C05480=1155.240,358.418,-80.283,-176.328,9.114,148.774
C05481=1155.245,358.171,-80.248,-176.331,9.110,148.773
C05482=1155.248,357.923,-80.214,-176.333,9.107,148.773
C05483=1155.252,357.676,-80.179,-176.336,9.102,148.773
C05484=1155.256,357.428,-80.144,-176.338,9.099,148.772
C05485=1155.261,357.181,-80.109,-176.341,9.095,148.772
C05486=1155.264,356.933,-80.075,-176.343,9.091,148.772
C05487=1155.268,356.685,-80.040,-176.345,9.087,148.771
C05488=1155.272,356.438,-80.005,-176.348,9.084,148.771
C05489=1155.276,356.190,-79.971,-176.350,9.080,148.771
C05490=1155.280,355.943,-79.937,-176.352,9.076,148.770
C05491=1155.284,355.695,-79.902,-176.355,9.072,148.770
C05492=1155.288,355.448,-79.868,-176.358,9.069,148.770
C05493=1155.292,355.200,-79.832,-176.360,9.065,148.770
C05494=1155.296,354.953,-79.798,-176.362,9.061,148.769
C05495=1155.299,354.705,-79.764,-176.365,9.057,148.769
C05496=1155.304,354.457,-79.729,-176.368,9.054,148.769
C05497=1155.308,354.210,-79.695,-176.370,9.049,148.768
C05498=1155.312,353.962,-79.660,-176.372,9.046,148.768
C05499=1155.316,353.715,-79.626,-176.375,9.042,148.768
C05500=1155.320,353.467,-79.592,-176.378,9.039,148.768
C05501=1155.324,353.220,-79.557,-176.380,9.034,148.767
C05502=1155.327,352.972,-79.523,-176.382,9.031,148.767
C05503=1155.332,352.724,-79.489,-176.385,9.027,148.767
C05504=1155.336,352.476,-79.454,-176.388,9.024,148.767
C05505=1155.340,352.229,-79.420,-176.390,9.019,148.766
C05506=1155.344,351.982,-79.385,-176.392,9.016,148.766
C05507=1155.348,351.734,-79.351,-176.395,9.012,148.766
C05508=1155.352,351.486,-79.317,-176.398,9.008,148.765
C05509=1155.355,351.239,-79.282,-176.400,9.004,148.765
C05510=1155.360,350.991,-79.248,-176.402,9.001,148.765
C05511=1155.364,350.744,-79.214,-176.405,8.997,148.764
C05512=1155.368,350.495,-79.180,-176.408,8.993,148.764
C05513=1155.372,350.248,-79.146,-176.410,8.989,148.764
C05514=1155.376,350.000,-79.111,-176.412,8.986,148.764
C05515=1155.380,349.753,-79.077,-176.415,8.982,148.763
C05516=1155.384,349.506,-79.043,-176.417,8.978,148.763
C05517=1155.388,349.257,-79.009,-176.420,8.974,148.763
C05518=1155.392,349.010,-78.976,-176.422,8.971,148.762
C05519=1155.396,348.763,-78.941,-176.425,8.967,148.762
C05520=1155.399,348.515,-78.907,-176.427,8.963,148.762
C05521=1155.404,348.267,-78.873,-176.430,8.960,148.762
C05522=1155.408,348.020,-78.839,-176.433,8.956,148.761
C05523=1155.411,347.772,-78.805,-176.435,8.952,148.761
C05524=1155.416,347.524,-78.771,-176.437,8.948,148.761
C05525=1155.420,347.277,-78.737,-176.440,8.945,148.761
C05526=1155.424,347.029,-78.703,-176.443,8.941,148.760
C05527=1155.428,346.781,-78.669,-176.445,8.938,148.760
C05528=1155.432,346.534,-78.635,-176.448,8.933,148.760
C05529=1155.436,346.286,-78.601,-176.450,8.930,148.759
C05530=1155.440,346.038,-78.567,-176.453,8.926,148.759
C05531=1155.444,345.791,-78.534,-176.455,8.922,148.759
C05532=1155.449,345.543,-78.500,-176.457,8.919,148.759
C05533=1155.452,345.295,-78.466,-176.460,8.915,148.759
C05534=1155.456,345.048,-78.432,-176.462,8.912,148.758
C05535=1155.461,344.800,-78.398,-176.465,8.907,148.758
C05536=1155.465,344.553,-78.364,-176.467,8.904,148.758
C05537=1155.468,344.304,-78.331,-176.470,8.900,148.757
C05538=1155.472,344.057,-78.297,-176.472,8.897,148.757
C05539=1155.477,343.809,-78.263,-176.475,8.893,148.757
C05540=1155.481,343.561,-78.230,-176.478,8.889,148.757
C05541=1155.484,343.314,-78.196,-176.480,8.886,148.757
C05542=1155.488,343.066,-78.162,-176.483,8.882,148.756
C05543=1155.493,342.818,-78.128,-176.485,8.879,148.756
C05544=1155.497,342.571,-78.095,-176.488,8.874,148.756
C05545=1155.501,342.323,-78.062,-176.490,8.871,148.755
C05546=1155.504,342.075,-78.027,-176.492,8.868,148.755
C05547=1155.509,341.827,-77.994,-176.495,8.864,148.755
C05548=1155.513,341.579,-77.961,-176.497,8.860,148.755
C05549=1155.517,341.332,-77.927,-176.500,8.856,148.755
C05550=1155.521,341.085,-77.894,-176.503,8.853,148.754
C05551=1155.526,340.837,-77.860,-176.505,8.850,148.754
C05552=1155.529,340.589,-77.826,-176.508,8.846,148.754
C05553=1155.533,340.341,-77.793,-176.510,8.842,148.754
C05554=1155.537,340.094,-77.760,-176.513,8.838,148.753
C05555=1155.542,339.814,-77.722,-176.516,8.834,148.753
C05556=1155.546,339.533,-77.684,-176.518,8.830,148.753
C05557=1155.551,339.254,-77.646,-176.521,8.826,148.752
C05558=1155.556,338.974,-77.609,-176.524,8.822,148.752
C05559=1155.560,338.727,-77.576,-176.527,8.818,148.752
C05560=1155.564,338.478,-77.541,-176.529,8.815,148.752
C05561=1155.568,338.230,-77.508,-176.532,8.811,148.752
C05562=1155.572,337.983,-77.474,-176.534,8.808,148.751
C05563=1155.576,337.735,-77.441,-176.536,8.804,148.751
C05564=1155.580,337.487,-77.408,-176.539,8.800,148.751
C05565=1155.584,337.240,-77.375,-176.542,8.797,148.751
C05566=1155.588,336.992,-77.342,-176.544,8.793,148.750
C05567=1155.593,336.744,-77.309,-176.547,8.790,148.750
C05568=1155.597,336.497,-77.275,-176.549,8.786,148.750
C05569=1155.600,336.248,-77.242,-176.552,8.782,148.750
C05570=1155.604,336.000,-77.209,-176.554,8.779,148.750
C05571=1155.608,335.753,-77.176,-176.557,8.776,148.749
C05572=1155.612,335.505,-77.143,-176.559,8.772,148.749
C05573=1155.616,335.258,-77.110,-176.562,8.768,148.749
C05574=1155.620,335.010,-77.077,-176.565,8.764,148.749
C05575=1155.624,334.762,-77.044,-176.567,8.761,148.749
C05576=1155.629,334.514,-77.010,-176.569,8.758,148.748
C05577=1155.633,334.267,-76.977,-176.572,8.753,148.748
C05578=1155.637,334.019,-76.944,-176.575,8.750,148.748
C05579=1155.641,333.771,-76.911,-176.577,8.747,148.748
C05580=1155.645,333.523,-76.879,-176.580,8.743,148.747
C05581=1155.649,333.275,-76.846,-176.582,8.740,148.747
C05582=1155.653,333.028,-76.813,-176.584,8.736,148.747
C05583=1155.657,332.780,-76.780,-176.587,8.732,148.747
C05584=1155.661,332.532,-76.747,-176.590,8.729,148.747
C05585=1155.665,332.284,-76.713,-176.592,8.726,148.746
C05586=1155.670,332.036,-76.681,-176.595,8.722,148.746
C05587=1155.673,331.789,-76.648,-176.597,8.718,148.746
C05588=1155.677,331.541,-76.615,-176.599,8.715,148.746
C05589=1155.681,331.293,-76.582,-176.603,8.711,148.746
C05590=1155.686,331.045,-76.550,-176.605,8.708,148.745
C05591=1155.690,330.797,-76.516,-176.608,8.704,148.745
C05592=1155.693,330.550,-76.484,-176.610,8.701,148.745
C05593=1155.698,330.301,-76.451,-176.613,8.697,148.745
C05594=1155.702,330.054,-76.418,-176.615,8.693,148.745
C05595=1155.706,329.806,-76.385,-176.618,8.690,148.744
C05596=1155.710,329.558,-76.353,-176.620,8.687,148.744
C05597=1155.714,329.310,-76.320,-176.622,8.683,148.744
C05598=1155.719,329.063,-76.287,-176.625,8.679,148.744
C05599=1155.723,328.815,-76.255,-176.628,8.676,148.744
C05600=1155.727,328.567,-76.222,-176.630,8.673,148.743
C05601=1155.731,328.319,-76.190,-176.633,8.669,148.743
C05602=1155.735,328.071,-76.157,-176.636,8.666,148.743
C05603=1155.739,327.824,-76.124,-176.638,8.662,148.743
C05604=1155.743,327.576,-76.092,-176.641,8.658,148.743
C05605=1155.747,327.328,-76.059,-176.643,8.655,148.743
C05606=1155.751,327.080,-76.027,-176.645,8.652,148.742
C05607=1155.756,326.833,-75.994,-176.648,8.648,148.742
C05608=1155.760,326.584,-75.962,-176.651,8.644,148.742
C05609=1155.763,326.337,-75.929,-176.653,8.641,148.742
C05610=1155.768,326.089,-75.897,-176.656,8.637,148.742
C05611=1155.772,325.841,-75.865,-176.658,8.634,148.741
C05612=1155.776,325.593,-75.832,-176.661,8.631,148.741
C05613=1155.780,325.344,-75.799,-176.663,8.627,148.741
C05614=1155.784,325.098,-75.767,-176.666,8.623,148.741
C05615=1155.789,324.849,-75.734,-176.668,8.620,148.741
C05616=1155.792,324.601,-75.703,-176.671,8.617,148.740
C05617=1155.796,324.354,-75.669,-176.674,8.613,148.740
C05618=1155.800,324.106,-75.638,-176.676,8.610,148.740
C05619=1155.805,323.857,-75.605,-176.679,8.606,148.740
C05620=1155.809,323.611,-75.573,-176.681,8.602,148.740
C05621=1155.813,323.362,-75.541,-176.684,8.599,148.740
C05622=1155.817,323.114,-75.509,-176.686,8.596,148.739
C05623=1155.821,322.866,-75.476,-176.689,8.593,148.739
C05624=1155.825,322.618,-75.444,-176.692,8.589,148.739
C05625=1155.830,322.371,-75.412,-176.694,8.585,148.739
C05626=1155.833,322.123,-75.380,-176.696,8.582,148.739
C05627=1155.838,321.874,-75.347,-176.699,8.578,148.739
C05628=1155.841,321.627,-75.315,-176.702,8.575,148.739
C05629=1155.846,321.380,-75.283,-176.704,8.572,148.738
C05630=1155.850,321.131,-75.251,-176.707,8.568,148.738
C05631=1155.854,320.883,-75.219,-176.710,8.564,148.738
C05632=1155.858,320.635,-75.187,-176.712,8.561,148.738
C05633=1155.862,320.388,-75.155,-176.715,8.558,148.738
C05634=1155.866,320.140,-75.123,-176.717,8.555,148.738
C05635=1155.870,319.892,-75.090,-176.720,8.551,148.737
C05636=1155.874,319.644,-75.058,-176.722,8.548,148.737
C05637=1155.879,319.396,-75.026,-176.725,8.545,148.737
C05638=1155.883,319.148,-74.994,-176.727,8.541,148.737
C05639=1155.886,318.900,-74.962,-176.730,8.537,148.737
C05640=1155.891,318.652,-74.930,-176.732,8.534,148.737
C05641=1155.895,318.404,-74.899,-176.735,8.531,148.736
C05642=1155.899,318.156,-74.867,-176.738,8.527,148.736
C05643=1155.903,317.908,-74.834,-176.740,8.524,148.736
C05644=1155.908,317.661,-74.803,-176.743,8.520,148.736
C05645=1155.911,317.413,-74.771,-176.745,8.517,148.736
C05646=1155.915,317.164,-74.739,-176.748,8.513,148.736
C05647=1155.920,316.917,-74.707,-176.751,8.510,148.736
C05648=1155.924,316.669,-74.675,-176.753,8.507,148.735
C05649=1155.927,316.421,-74.643,-176.756,8.504,148.735
C05650=1155.932,316.173,-74.613,-176.759,8.500,148.735
C05651=1155.937,315.924,-74.580,-176.761,8.496,148.735
C05652=1155.941,315.677,-74.549,-176.763,8.493,148.735
C05653=1155.945,315.429,-74.517,-176.766,8.490,148.735
C05654=1155.948,315.181,-74.485,-176.768,8.487,148.735
C05655=1155.953,314.933,-74.453,-176.771,8.483,148.734
C05656=1155.957,314.685,-74.422,-176.773,8.479,148.734
C05657=1155.961,314.437,-74.390,-176.776,8.476,148.734
C05658=1155.965,314.189,-74.358,-176.778,8.473,148.734
C05659=1155.970,313.912,-74.323,-176.781,8.469,148.734
C05660=1155.975,313.635,-74.288,-176.785,8.465,148.734
C05661=1155.979,313.357,-74.253,-176.788,8.461,148.734
C05662=1155.984,313.079,-74.217,-176.790,8.458,148.733
C05663=1155.988,312.832,-74.186,-176.793,8.454,148.733
C05664=1155.992,312.584,-74.153,-176.796,8.451,148.733
C05665=1155.997,312.336,-74.122,-176.798,8.448,148.733
C05666=1156.001,312.088,-74.091,-176.801,8.445,148.733
C05667=1156.005,311.840,-74.059,-176.803,8.441,148.733
C05668=1156.009,311.592,-74.028,-176.806,8.437,148.733
C05669=1156.013,311.344,-73.996,-176.809,8.434,148.733
C05670=1156.017,311.096,-73.965,-176.811,8.431,148.732
C05671=1156.022,310.848,-73.934,-176.813,8.428,148.732
C05672=1156.025,310.600,-73.902,-176.816,8.425,148.732
C05673=1156.030,310.352,-73.871,-176.819,8.421,148.732
C05674=1156.034,310.104,-73.839,-176.821,8.417,148.732
C05675=1156.038,309.856,-73.808,-176.824,8.414,148.732
C05676=1156.042,309.608,-73.777,-176.826,8.411,148.732
C05677=1156.047,309.360,-73.745,-176.829,8.408,148.732
C05678=1156.051,309.112,-73.714,-176.832,8.404,148.731
C05679=1156.056,308.864,-73.683,-176.834,8.401,148.731
C05680=1156.059,308.616,-73.651,-176.837,8.398,148.731
C05681=1156.064,308.368,-73.620,-176.839,8.395,148.731
C05682=1156.067,308.120,-73.590,-176.842,8.391,148.731
C05683=1156.071,307.872,-73.558,-176.845,8.388,148.731
C05684=1156.075,307.624,-73.527,-176.847,8.384,148.731
C05685=1156.080,307.376,-73.496,-176.850,8.381,148.731
C05686=1156.084,307.128,-73.464,-176.852,8.378,148.731
C05687=1156.088,306.880,-73.434,-176.855,8.375,148.730
C05688=1156.092,306.632,-73.402,-176.858,8.371,148.730
C05689=1156.097,306.384,-73.371,-176.860,8.368,148.730
C05690=1156.101,306.136,-73.340,-176.863,8.365,148.730
C05691=1156.105,305.888,-73.308,-176.865,8.361,148.730
C05692=1156.110,305.640,-73.278,-176.868,8.358,148.730
C05693=1156.114,305.391,-73.247,-176.871,8.354,148.730
C05694=1156.118,305.144,-73.215,-176.873,8.351,148.730
C05695=1156.122,304.896,-73.185,-176.876,8.348,148.730
C05696=1156.126,304.647,-73.154,-176.878,8.345,148.729
C05697=1156.130,304.400,-73.123,-176.881,8.342,148.729
C05698=1156.134,304.151,-73.092,-176.883,8.339,148.729
C05699=1156.139,303.904,-73.060,-176.886,8.335,148.729
C05700=1156.143,303.656,-73.030,-176.889,8.332,148.729
C05701=1156.147,303.407,-72.999,-176.891,8.328,148.729
C05702=1156.151,303.159,-72.968,-176.894,8.325,148.729
C05703=1156.156,302.911,-72.938,-176.896,8.322,148.729
C05704=1156.160,302.663,-72.906,-176.899,8.319,148.729
C05705=1156.164,302.415,-72.875,-176.902,8.315,148.729
C05706=1156.168,302.168,-72.845,-176.904,8.312,148.728
C05707=1156.172,301.919,-72.814,-176.907,8.309,148.728
C05708=1156.177,301.671,-72.783,-176.909,8.306,148.728
C05709=1156.181,301.423,-72.752,-176.912,8.303,148.728
C05710=1156.185,301.175,-72.722,-176.915,8.299,148.728
C05711=1156.189,300.927,-72.691,-176.917,8.296,148.728
C05712=1156.194,300.679,-72.660,-176.920,8.292,148.728
C05713=1156.197,300.430,-72.630,-176.923,8.289,148.728
C05714=1156.202,300.183,-72.599,-176.925,8.286,148.728
C05715=1156.206,299.935,-72.568,-176.928,8.283,148.728
C05716=1156.210,299.687,-72.538,-176.930,8.280,148.728
C05717=1156.214,299.438,-72.507,-176.933,8.277,148.728
C05718=1156.219,299.190,-72.476,-176.935,8.274,148.727
C05719=1156.223,298.943,-72.446,-176.939,8.270,148.727
C05720=1156.227,298.695,-72.415,-176.941,8.266,148.727
C05721=1156.232,298.445,-72.385,-176.944,8.263,148.727
C05722=1156.236,298.198,-72.354,-176.946,8.260,148.727
C05723=1156.240,297.950,-72.324,-176.949,8.257,148.727
C05724=1156.245,297.702,-72.293,-176.951,8.254,148.727
C05725=1156.248,297.453,-72.262,-176.954,8.251,148.727
C05726=1156.253,297.206,-72.232,-176.957,8.247,148.727
C05727=1156.257,296.957,-72.202,-176.960,8.244,148.727
C05728=1156.261,296.709,-72.171,-176.962,8.241,148.727
C05729=1156.265,296.461,-72.141,-176.965,8.238,148.727
C05730=1156.269,296.213,-72.110,-176.967,8.234,148.727
C05731=1156.273,295.965,-72.080,-176.970,8.232,148.727
C05732=1156.278,295.717,-72.050,-176.972,8.228,148.726
C05733=1156.283,295.469,-72.019,-176.975,8.225,148.726
C05734=1156.286,295.220,-71.989,-176.978,8.222,148.726
C05735=1156.291,294.972,-71.959,-176.980,8.218,148.726
C05736=1156.295,294.724,-71.928,-176.983,8.215,148.726
C05737=1156.299,294.477,-71.898,-176.986,8.212,148.726
C05738=1156.304,294.228,-71.868,-176.988,8.209,148.726
C05739=1156.307,293.980,-71.838,-176.991,8.206,148.726
C05740=1156.311,293.732,-71.807,-176.993,8.203,148.726
C05741=1156.316,293.483,-71.777,-176.996,8.200,148.726
C05742=1156.320,293.235,-71.747,-176.998,8.197,148.726
C05743=1156.324,292.988,-71.716,-177.002,8.193,148.726
C05744=1156.329,292.739,-71.686,-177.004,8.190,148.726
C05745=1156.333,292.492,-71.656,-177.007,8.187,148.726
C05746=1156.337,292.243,-71.626,-177.009,8.183,148.726
C05747=1156.341,291.995,-71.596,-177.012,8.180,148.726
C05748=1156.345,291.746,-71.566,-177.014,8.177,148.725
C05749=1156.350,291.498,-71.535,-177.017,8.174,148.725
C05750=1156.354,291.250,-71.506,-177.020,8.171,148.725
C05751=1156.358,291.003,-71.476,-177.022,8.168,148.725
C05752=1156.363,290.754,-71.446,-177.025,8.165,148.725
C05753=1156.367,290.506,-71.416,-177.028,8.161,148.725
C05754=1156.371,290.258,-71.386,-177.030,8.158,148.725
C05755=1156.375,290.009,-71.355,-177.033,8.155,148.725
C05756=1156.379,289.761,-71.326,-177.036,8.152,148.725
C05757=1156.383,289.513,-71.296,-177.038,8.149,148.725
C05758=1156.388,289.265,-71.265,-177.041,8.146,148.725
C05759=1156.392,289.017,-71.236,-177.043,8.142,148.725
C05760=1156.396,288.769,-71.206,-177.046,8.139,148.725
C05761=1156.400,288.521,-71.176,-177.048,8.136,148.725
C05762=1156.405,288.272,-71.146,-177.051,8.133,148.725
C05763=1156.410,287.997,-71.113,-177.055,8.129,148.725
C05764=1156.415,287.722,-71.080,-177.057,8.126,148.725
C05765=1156.419,287.447,-71.047,-177.060,8.122,148.725
C05766=1156.424,287.172,-71.014,-177.063,8.119,148.725
C05767=1156.428,286.924,-70.984,-177.066,8.117,148.725
C05768=1156.432,286.676,-70.955,-177.068,8.113,148.725
C05769=1156.437,286.428,-70.925,-177.071,8.109,148.725
C05770=1156.441,286.179,-70.895,-177.074,8.107,148.725
C05771=1156.446,285.931,-70.866,-177.076,8.103,148.724
C05772=1156.450,285.683,-70.836,-177.079,8.100,148.724
C05773=1156.454,285.435,-70.806,-177.082,8.097,148.725
C05774=1156.458,285.187,-70.777,-177.084,8.094,148.724
C05775=1156.462,284.938,-70.747,-177.087,8.091,148.724
C05776=1156.467,284.690,-70.717,-177.090,8.088,148.724
C05777=1156.471,284.442,-70.688,-177.092,8.085,148.724
C05778=1156.475,284.193,-70.658,-177.095,8.082,148.724
C05779=1156.479,283.946,-70.628,-177.098,8.079,148.724
C05780=1156.483,283.697,-70.599,-177.100,8.076,148.724
C05781=1156.488,283.449,-70.569,-177.103,8.073,148.724
C05782=1156.492,283.201,-70.540,-177.105,8.070,148.724
C05783=1156.496,282.953,-70.510,-177.108,8.067,148.724
C05784=1156.500,282.704,-70.481,-177.111,8.064,148.724
C05785=1156.505,282.456,-70.451,-177.113,8.061,148.724
C05786=1156.509,282.207,-70.421,-177.116,8.057,148.724
C05787=1156.513,281.959,-70.392,-177.118,8.054,148.724
C05788=1156.518,281.712,-70.363,-177.122,8.051,148.724
C05789=1156.522,281.463,-70.333,-177.124,8.048,148.724
C05790=1156.527,281.215,-70.304,-177.127,8.044,148.724
C05791=1156.531,280.967,-70.275,-177.130,8.041,148.724
C05792=1156.535,280.718,-70.246,-177.132,8.038,148.724
C05793=1156.539,280.470,-70.216,-177.135,8.036,148.724
C05794=1156.544,280.221,-70.187,-177.137,8.032,148.724
C05795=1156.548,279.973,-70.157,-177.140,8.029,148.724
C05796=1156.553,279.726,-70.128,-177.143,8.026,148.724
C05797=1156.557,279.477,-70.099,-177.145,8.023,148.724
C05798=1156.561,279.229,-70.069,-177.148,8.020,148.724
C05799=1156.565,278.981,-70.040,-177.151,8.017,148.724
C05800=1156.569,278.732,-70.012,-177.154,8.014,148.724
C05801=1156.573,278.484,-69.982,-177.156,8.011,148.724
C05802=1156.578,278.236,-69.953,-177.159,8.008,148.724
C05803=1156.582,277.988,-69.924,-177.161,8.005,148.724
C05804=1156.586,277.739,-69.895,-177.164,8.002,148.724
C05805=1156.591,277.491,-69.866,-177.166,7.999,148.724
C05806=1156.595,277.243,-69.836,-177.169,7.996,148.724
C05807=1156.599,276.994,-69.807,-177.172,7.993,148.724
C05808=1156.604,276.746,-69.778,-177.175,7.990,148.724
C05809=1156.608,276.498,-69.749,-177.177,7.987,148.724
C05810=1156.612,276.250,-69.720,-177.180,7.984,148.724
C05811=1156.616,276.001,-69.691,-177.183,7.981,148.724
C05812=1156.620,275.753,-69.662,-177.185,7.978,148.724
C05813=1156.625,275.505,-69.633,-177.188,7.975,148.724
C05814=1156.629,275.257,-69.605,-177.190,7.972,148.724
C05815=1156.633,275.008,-69.575,-177.193,7.969,148.724
C05816=1156.638,274.759,-69.546,-177.196,7.966,148.724
C05817=1156.642,274.512,-69.517,-177.199,7.963,148.724
C05818=1156.647,274.264,-69.488,-177.201,7.960,148.724
C05819=1156.650,274.015,-69.460,-177.204,7.957,148.724
C05820=1156.654,273.767,-69.430,-177.207,7.954,148.724
C05821=1156.660,273.519,-69.402,-177.209,7.951,148.724
C05822=1156.664,273.270,-69.372,-177.212,7.948,148.724
C05823=1156.668,273.022,-69.344,-177.215,7.945,148.724
C05824=1156.672,272.774,-69.315,-177.218,7.942,148.724
C05825=1156.677,272.525,-69.287,-177.220,7.939,148.724
C05826=1156.680,272.277,-69.258,-177.223,7.936,148.724
C05827=1156.685,272.029,-69.229,-177.225,7.933,148.724
C05828=1156.690,271.780,-69.201,-177.228,7.930,148.724
C05829=1156.694,271.532,-69.171,-177.231,7.927,148.724
C05830=1156.698,271.283,-69.143,-177.234,7.924,148.724
C05831=1156.703,271.036,-69.114,-177.236,7.921,148.724
C05832=1156.706,270.787,-69.086,-177.239,7.918,148.724
C05833=1156.711,270.538,-69.057,-177.242,7.915,148.724
C05834=1156.716,270.291,-69.028,-177.244,7.912,148.724
C05835=1156.719,270.042,-69.000,-177.247,7.909,148.724
C05836=1156.724,269.794,-68.971,-177.250,7.906,148.724
C05837=1156.729,269.546,-68.942,-177.252,7.902,148.724
C05838=1156.732,269.297,-68.914,-177.255,7.900,148.724
C05839=1156.737,269.049,-68.885,-177.258,7.897,148.724
C05840=1156.741,268.800,-68.857,-177.260,7.894,148.724
C05841=1156.745,268.552,-68.828,-177.263,7.891,148.724
C05842=1156.750,268.304,-68.799,-177.265,7.889,148.724
C05843=1156.754,268.055,-68.771,-177.268,7.886,148.724
C05844=1156.759,267.807,-68.743,-177.271,7.883,148.725
C05845=1156.763,267.559,-68.714,-177.273,7.879,148.724
C05846=1156.767,267.310,-68.685,-177.276,7.876,148.724
C05847=1156.772,267.063,-68.658,-177.279,7.874,148.724
C05848=1156.776,266.814,-68.629,-177.282,7.871,148.725
C05849=1156.780,266.566,-68.601,-177.284,7.868,148.725
C05850=1156.785,266.317,-68.572,-177.287,7.865,148.725
C05851=1156.789,266.070,-68.544,-177.290,7.862,148.725
C05852=1156.793,265.821,-68.515,-177.293,7.859,148.725
C05853=1156.797,265.572,-68.487,-177.295,7.856,148.725
C05854=1156.802,265.324,-68.459,-177.298,7.853,148.725
C05855=1156.806,265.075,-68.430,-177.301,7.850,148.725
C05856=1156.811,264.827,-68.402,-177.303,7.847,148.725
C05857=1156.815,264.579,-68.374,-177.306,7.844,148.725
C05858=1156.820,264.330,-68.346,-177.309,7.841,148.725
C05859=1156.824,264.082,-68.317,-177.312,7.838,148.725
C05860=1156.828,263.834,-68.290,-177.314,7.835,148.725
C05861=1156.832,263.585,-68.261,-177.317,7.833,148.725
C05862=1156.837,263.337,-68.233,-177.319,7.830,148.725
C05863=1156.841,263.088,-68.204,-177.322,7.827,148.725
C05864=1156.846,262.840,-68.177,-177.325,7.824,148.725
C05865=1156.849,262.592,-68.148,-177.328,7.821,148.725
C05866=1156.855,262.344,-68.120,-177.330,7.818,148.725
C05867=1156.859,262.070,-68.089,-177.333,7.815,148.725
C05868=1156.864,261.797,-68.059,-177.337,7.811,148.725
C05869=1156.869,261.524,-68.028,-177.339,7.808,148.725
C05870=1156.873,261.250,-67.997,-177.342,7.805,148.726
C05871=1156.878,261.002,-67.969,-177.345,7.802,148.726
C05872=1156.882,260.754,-67.941,-177.348,7.800,148.726
C05873=1156.886,260.506,-67.913,-177.350,7.797,148.726
C05874=1156.891,260.257,-67.884,-177.353,7.794,148.726
C05875=1156.896,260.008,-67.857,-177.356,7.791,148.726
C05876=1156.899,259.760,-67.829,-177.359,7.788,148.726
C05877=1156.904,259.512,-67.801,-177.361,7.785,148.726
C05878=1156.908,259.263,-67.773,-177.364,7.782,148.726
C05879=1156.913,259.015,-67.746,-177.366,7.779,148.726
C05880=1156.917,258.767,-67.718,-177.369,7.776,148.726
C05881=1156.921,258.518,-67.690,-177.371,7.774,148.726
C05882=1156.926,258.269,-67.662,-177.374,7.771,148.726
C05883=1156.930,258.021,-67.634,-177.377,7.768,148.726
C05884=1156.934,257.773,-67.606,-177.380,7.765,148.726
C05885=1156.939,257.524,-67.579,-177.383,7.762,148.726
C05886=1156.943,257.276,-67.551,-177.385,7.759,148.726
C05887=1156.948,257.028,-67.522,-177.388,7.756,148.726
C05888=1156.952,256.778,-67.495,-177.391,7.753,148.726
C05889=1156.956,256.530,-67.467,-177.393,7.751,148.727
C05890=1156.961,256.283,-67.439,-177.396,7.748,148.727
C05891=1156.965,256.033,-67.412,-177.399,7.745,148.727
C05892=1156.969,255.786,-67.384,-177.401,7.742,148.727
C05893=1156.974,255.537,-67.357,-177.404,7.739,148.727
C05894=1156.978,255.288,-67.328,-177.407,7.736,148.727
C05895=1156.983,255.040,-67.301,-177.410,7.733,148.727
C05896=1156.987,254.792,-67.274,-177.412,7.730,148.727
C05897=1156.991,254.543,-67.246,-177.415,7.728,148.727
C05898=1156.996,254.295,-67.218,-177.418,7.725,148.727
C05899=1157.000,254.046,-67.191,-177.421,7.722,148.727
C05900=1157.005,253.798,-67.164,-177.423,7.720,148.728
C05901=1157.009,253.549,-67.136,-177.426,7.717,148.728
C05902=1157.013,253.301,-67.108,-177.429,7.714,148.728
C05903=1157.018,253.053,-67.081,-177.432,7.711,148.728
C05904=1157.022,252.804,-67.054,-177.434,7.708,148.728
C05905=1157.026,252.556,-67.026,-177.437,7.706,148.728
C05906=1157.031,252.307,-66.999,-177.439,7.703,148.728
C05907=1157.035,252.059,-66.971,-177.442,7.700,148.728
C05908=1157.039,251.810,-66.944,-177.445,7.697,148.728
C05909=1157.044,251.562,-66.917,-177.448,7.694,148.728
C05910=1157.048,251.314,-66.889,-177.451,7.691,148.728
C05911=1157.053,251.065,-66.862,-177.453,7.688,148.728
C05912=1157.057,250.816,-66.835,-177.456,7.686,148.728
C05913=1157.061,250.568,-66.807,-177.458,7.683,148.728
C05914=1157.066,250.320,-66.780,-177.461,7.680,148.728
C05915=1157.070,250.071,-66.753,-177.464,7.677,148.729
C05916=1157.075,249.822,-66.725,-177.467,7.674,148.729
C05917=1157.079,249.574,-66.697,-177.470,7.672,148.729
C05918=1157.084,249.326,-66.670,-177.472,7.669,148.729
C05919=1157.088,249.077,-66.643,-177.475,7.666,148.729
C05920=1157.092,248.829,-66.617,-177.478,7.664,148.729
C05921=1157.096,248.580,-66.589,-177.480,7.661,148.729
C05922=1157.101,248.332,-66.562,-177.483,7.658,148.729
C05923=1157.105,248.083,-66.535,-177.486,7.655,148.729
C05924=1157.110,247.835,-66.508,-177.488,7.653,148.729
C05925=1157.115,247.586,-66.480,-177.491,7.650,148.730
C05926=1157.119,247.338,-66.453,-177.494,7.647,148.730
C05927=1157.122,247.089,-66.427,-177.497,7.644,148.730
C05928=1157.127,246.841,-66.399,-177.500,7.641,148.730
C05929=1157.132,246.592,-66.372,-177.502,7.638,148.730
C05930=1157.136,246.344,-66.345,-177.505,7.636,148.730
C05931=1157.141,246.095,-66.318,-177.507,7.633,148.730
C05932=1157.145,245.847,-66.291,-177.510,7.630,148.730
C05933=1157.149,245.599,-66.264,-177.513,7.627,148.730
C05934=1157.153,245.350,-66.237,-177.516,7.624,148.730
C05935=1157.158,245.101,-66.210,-177.518,7.623,148.731
C05936=1157.162,244.853,-66.183,-177.521,7.620,148.731
C05937=1157.167,244.605,-66.156,-177.524,7.617,148.731
C05938=1157.172,244.355,-66.130,-177.527,7.614,148.731
C05939=1157.176,244.107,-66.103,-177.529,7.611,148.731
C05940=1157.180,243.859,-66.076,-177.532,7.609,148.731
C05941=1157.185,243.610,-66.049,-177.534,7.606,148.731
C05942=1157.190,243.362,-66.022,-177.538,7.603,148.731
C05943=1157.193,243.113,-65.995,-177.540,7.600,148.732
C05944=1157.197,242.864,-65.968,-177.543,7.597,148.732
C05945=1157.202,242.616,-65.941,-177.545,7.595,148.732
C05946=1157.207,242.367,-65.914,-177.548,7.592,148.732
C05947=1157.211,242.119,-65.888,-177.551,7.589,148.732
C05948=1157.216,241.870,-65.861,-177.554,7.586,148.732
C05949=1157.220,241.622,-65.835,-177.557,7.584,148.732
C05950=1157.224,241.373,-65.808,-177.559,7.582,148.732
C05951=1157.229,241.125,-65.781,-177.562,7.579,148.732
C05952=1157.233,240.877,-65.754,-177.565,7.576,148.732
C05953=1157.238,240.628,-65.728,-177.567,7.573,148.733
C05954=1157.242,240.379,-65.701,-177.570,7.570,148.733
C05955=1157.246,240.131,-65.674,-177.573,7.568,148.733
C05956=1157.251,239.883,-65.647,-177.576,7.565,148.733
C05957=1157.255,239.634,-65.621,-177.578,7.562,148.733
C05958=1157.260,239.385,-65.594,-177.581,7.559,148.733
C05959=1157.264,239.137,-65.568,-177.583,7.557,148.733
C05960=1157.269,238.888,-65.542,-177.587,7.554,148.734
C05961=1157.273,238.639,-65.515,-177.589,7.552,148.734
C05962=1157.277,238.391,-65.488,-177.592,7.549,148.734
C05963=1157.282,238.142,-65.462,-177.594,7.546,148.734
C05964=1157.286,237.894,-65.435,-177.597,7.544,148.734
C05965=1157.291,237.645,-65.409,-177.600,7.541,148.734
C05966=1157.295,237.397,-65.382,-177.603,7.538,148.734
C05967=1157.300,237.148,-65.355,-177.605,7.536,148.734
C05968=1157.304,236.899,-65.330,-177.608,7.533,148.734
C05969=1157.309,236.651,-65.303,-177.611,7.530,148.735
C05970=1157.313,236.402,-65.277,-177.614,7.527,148.735
C05971=1157.318,236.130,-65.247,-177.617,7.524,148.735
C05972=1157.322,235.859,-65.219,-177.620,7.522,148.735
C05973=1157.328,235.587,-65.190,-177.623,7.519,148.735
C05974=1157.332,235.316,-65.161,-177.626,7.516,148.735
C05975=1157.336,235.067,-65.136,-177.629,7.513,148.735
C05976=1157.341,234.818,-65.109,-177.631,7.510,148.736
C05977=1157.346,234.570,-65.083,-177.634,7.508,148.736
C05978=1157.351,234.322,-65.056,-177.637,7.505,148.736
C05979=1157.355,234.073,-65.030,-177.640,7.502,148.736
C05980=1157.359,233.824,-65.005,-177.642,7.500,148.736
C05981=1157.364,233.576,-64.978,-177.645,7.498,148.736
C05982=1157.368,233.327,-64.952,-177.648,7.495,148.737
C05983=1157.372,233.079,-64.925,-177.651,7.492,148.737
C05984=1157.377,232.830,-64.899,-177.653,7.490,148.737
C05985=1157.382,232.581,-64.874,-177.656,7.487,148.737
C05986=1157.386,232.333,-64.847,-177.659,7.484,148.737
C05987=1157.391,232.084,-64.821,-177.662,7.481,148.737
C05988=1157.395,231.835,-64.795,-177.664,7.479,148.737
C05989=1157.399,231.587,-64.769,-177.667,7.477,148.738
C05990=1157.404,231.338,-64.742,-177.670,7.474,148.738
C05991=1157.408,231.090,-64.717,-177.672,7.472,148.738
C05992=1157.413,230.841,-64.691,-177.675,7.469,148.738
C05993=1157.418,230.592,-64.665,-177.678,7.466,148.738
C05994=1157.422,230.344,-64.638,-177.681,7.463,148.738
C05995=1157.426,230.095,-64.612,-177.683,7.461,148.738
C05996=1157.431,229.847,-64.587,-177.686,7.458,148.739
C05997=1157.436,229.598,-64.561,-177.689,7.455,148.739
C05998=1157.439,229.350,-64.534,-177.691,7.453,148.739
C05999=1157.444,229.101,-64.509,-177.694,7.451,148.739
C06000=1157.448,228.852,-64.483,-177.697,7.448,148.739
C06001=1157.453,228.604,-64.457,-177.699,7.446,148.739
C06002=1157.458,228.355,-64.431,-177.702,7.443,148.739
C06003=1157.462,228.106,-64.405,-177.705,7.440,148.740
C06004=1157.466,227.857,-64.380,-177.708,7.438,148.740
C06005=1157.471,227.609,-64.354,-177.710,7.435,148.740
C06006=1157.475,227.360,-64.328,-177.714,7.432,148.740
C06007=1157.479,227.112,-64.302,-177.716,7.430,148.740
C06008=1157.483,226.863,-64.276,-177.719,7.427,148.740
C06009=1157.489,226.615,-64.250,-177.722,7.425,148.741
C06010=1157.493,226.366,-64.224,-177.725,7.422,148.741
C06011=1157.497,226.117,-64.199,-177.727,7.420,148.741
C06012=1157.502,225.868,-64.173,-177.730,7.417,148.741
C06013=1157.506,225.620,-64.148,-177.733,7.414,148.741
C06014=1157.511,225.372,-64.122,-177.735,7.412,148.741
C06015=1157.515,225.123,-64.096,-177.738,7.409,148.741
C06016=1157.520,224.875,-64.071,-177.741,7.407,148.742
C06017=1157.524,224.625,-64.046,-177.743,7.404,148.742
C06018=1157.528,224.376,-64.020,-177.746,7.402,148.742
C06019=1157.533,224.128,-63.995,-177.749,7.399,148.742
C06020=1157.538,223.879,-63.969,-177.752,7.397,148.742
C06021=1157.542,223.630,-63.942,-177.755,7.394,148.743
C06022=1157.547,223.382,-63.917,-177.758,7.391,148.743
C06023=1157.552,223.133,-63.891,-177.760,7.389,148.743
C06024=1157.556,222.885,-63.866,-177.763,7.387,148.743
C06025=1157.561,222.636,-63.841,-177.765,7.384,148.743
C06026=1157.565,222.387,-63.815,-177.768,7.382,148.743
C06027=1157.569,222.138,-63.789,-177.771,7.379,148.744
C06028=1157.574,221.890,-63.764,-177.773,7.377,148.744
C06029=1157.578,221.642,-63.739,-177.776,7.374,148.744
C06030=1157.583,221.393,-63.714,-177.779,7.371,148.744
C06031=1157.587,221.144,-63.688,-177.782,7.369,148.744
C06032=1157.591,220.895,-63.663,-177.784,7.366,148.744
C06033=1157.596,220.647,-63.637,-177.788,7.364,148.745
C06034=1157.601,220.398,-63.612,-177.790,7.362,148.745
C06035=1157.605,220.150,-63.587,-177.793,7.359,148.745
C06036=1157.610,219.901,-63.561,-177.795,7.357,148.745
C06037=1157.614,219.652,-63.536,-177.798,7.354,148.745
C06038=1157.619,219.403,-63.511,-177.801,7.351,148.746
C06039=1157.623,219.155,-63.485,-177.804,7.349,148.746
C06040=1157.628,218.906,-63.461,-177.806,7.346,148.746
C06041=1157.632,218.657,-63.435,-177.809,7.345,148.746
C06042=1157.637,218.409,-63.410,-177.812,7.342,148.746
C06043=1157.641,218.160,-63.385,-177.815,7.339,148.747
C06044=1157.645,217.911,-63.359,-177.817,7.337,148.747
C06045=1157.651,217.662,-63.334,-177.820,7.334,148.747
C06046=1157.654,217.414,-63.309,-177.823,7.331,148.747
C06047=1157.659,217.166,-63.284,-177.826,7.329,148.747
C06048=1157.663,216.916,-63.259,-177.829,7.327,148.748
C06049=1157.668,216.668,-63.233,-177.831,7.325,148.748
C06050=1157.673,216.419,-63.208,-177.834,7.322,148.748
C06051=1157.677,216.171,-63.183,-177.836,7.320,148.748
C06052=1157.681,215.922,-63.158,-177.839,7.317,148.748
C06053=1157.686,215.673,-63.133,-177.842,7.314,148.749
C06054=1157.691,215.424,-63.108,-177.845,7.312,148.749
C06055=1157.695,215.176,-63.083,-177.847,7.309,148.749
C06056=1157.699,214.927,-63.058,-177.850,7.308,148.749
C06057=1157.704,214.678,-63.034,-177.853,7.305,148.749
C06058=1157.709,214.429,-63.008,-177.856,7.302,148.750
C06059=1157.713,214.181,-62.984,-177.858,7.300,148.750
C06060=1157.717,213.932,-62.958,-177.862,7.297,148.750
C06061=1157.722,213.683,-62.933,-177.864,7.295,148.750
C06062=1157.726,213.434,-62.909,-177.867,7.292,148.750
C06063=1157.731,213.186,-62.883,-177.869,7.291,148.751
C06064=1157.736,212.937,-62.859,-177.872,7.288,148.751
C06065=1157.740,212.688,-62.834,-177.875,7.285,148.751
C06066=1157.745,212.440,-62.809,-177.878,7.283,148.751
C06067=1157.749,212.191,-62.784,-177.881,7.280,148.751
C06068=1157.754,211.942,-62.760,-177.883,7.278,148.751
C06069=1157.758,211.694,-62.734,-177.886,7.276,148.752
C06070=1157.763,211.445,-62.709,-177.888,7.273,148.752
C06071=1157.767,211.196,-62.685,-177.891,7.271,148.752
C06072=1157.772,210.947,-62.660,-177.894,7.269,148.752
C06073=1157.776,210.699,-62.636,-177.897,7.266,148.752
C06074=1157.781,210.450,-62.611,-177.900,7.263,148.753
C06075=1157.786,210.180,-62.584,-177.902,7.261,148.753
C06076=1157.791,209.909,-62.557,-177.905,7.259,148.753
C06077=1157.795,209.639,-62.530,-177.909,7.256,148.754
C06078=1157.801,209.368,-62.503,-177.911,7.253,148.754
C06079=1157.805,209.119,-62.478,-177.914,7.251,148.754
C06080=1157.810,208.871,-62.454,-177.917,7.248,148.754
C06081=1157.815,208.622,-62.430,-177.920,7.246,148.754
C06082=1157.818,208.373,-62.405,-177.922,7.244,148.755
C06083=1157.824,208.124,-62.380,-177.926,7.241,148.755
C06084=1157.828,207.876,-62.356,-177.928,7.239,148.755
C06085=1157.833,207.626,-62.331,-177.931,7.236,148.755
C06086=1157.837,207.378,-62.307,-177.933,7.234,148.755
C06087=1157.842,207.129,-62.283,-177.937,7.232,148.756
C06088=1157.846,206.881,-62.257,-177.939,7.230,148.756
C06089=1157.851,206.632,-62.233,-177.942,7.227,148.756
C06090=1157.855,206.383,-62.209,-177.944,7.225,148.756
C06091=1157.860,206.134,-62.184,-177.947,7.222,148.757
C06092=1157.864,205.886,-62.160,-177.950,7.220,148.757
C06093=1157.869,205.637,-62.135,-177.953,7.218,148.757
C06094=1157.874,205.388,-62.112,-177.955,7.216,148.757
C06095=1157.878,205.139,-62.087,-177.958,7.213,148.758
C06096=1157.883,204.890,-62.062,-177.961,7.211,148.758
C06097=1157.887,204.642,-62.038,-177.964,7.208,148.758
C06098=1157.892,204.393,-62.014,-177.966,7.206,148.758
C06099=1157.896,204.144,-61.989,-177.969,7.204,148.758
C06100=1157.900,203.895,-61.965,-177.971,7.201,148.759
C06101=1157.906,203.647,-61.940,-177.975,7.199,148.759
C06102=1157.910,203.398,-61.916,-177.977,7.197,148.759
C06103=1157.914,203.149,-61.892,-177.980,7.194,148.759
C06104=1157.919,202.900,-61.868,-177.982,7.192,148.759
C06105=1157.924,202.651,-61.844,-177.986,7.189,148.760
C06106=1157.928,202.403,-61.820,-177.988,7.187,148.760
C06107=1157.933,202.153,-61.795,-177.991,7.185,148.760
C06108=1157.937,201.905,-61.771,-177.993,7.183,148.760
C06109=1157.942,201.656,-61.747,-177.997,7.180,148.761
C06110=1157.947,201.407,-61.723,-177.999,7.178,148.761
C06111=1157.951,201.159,-61.699,-178.002,7.175,148.761
C06112=1157.955,200.910,-61.674,-178.005,7.174,148.761
C06113=1157.960,200.661,-61.651,-178.008,7.171,148.762
C06114=1157.965,200.412,-61.626,-178.010,7.169,148.762
C06115=1157.969,200.164,-61.602,-178.013,7.166,148.762
C06116=1157.974,199.915,-61.578,-178.016,7.164,148.762
C06117=1157.978,199.665,-61.554,-178.018,7.161,148.762
C06118=1157.983,199.417,-61.530,-178.021,7.160,148.763
C06119=1157.987,199.168,-61.506,-178.023,7.158,148.763
C06120=1157.992,198.919,-61.482,-178.027,7.155,148.763
C06121=1157.996,198.671,-61.458,-178.029,7.153,148.764
C06122=1158.001,198.422,-61.435,-178.032,7.150,148.764
C06123=1158.006,198.173,-61.410,-178.035,7.148,148.764
C06124=1158.010,197.924,-61.386,-178.038,7.146,148.764
C06125=1158.015,197.675,-61.362,-178.040,7.144,148.765
C06126=1158.019,197.427,-61.338,-178.043,7.141,148.765
C06127=1158.024,197.178,-61.315,-178.046,7.139,148.765
C06128=1158.028,196.929,-61.291,-178.049,7.137,148.765
C06129=1158.033,196.680,-61.267,-178.051,7.134,148.765
C06130=1158.038,196.431,-61.243,-178.054,7.133,148.766
C06131=1158.042,196.183,-61.219,-178.057,7.130,148.766
C06132=1158.047,195.934,-61.195,-178.059,7.128,148.766
C06133=1158.051,195.685,-61.171,-178.063,7.125,148.767
C06134=1158.056,195.436,-61.148,-178.065,7.123,148.767
C06135=1158.060,195.187,-61.124,-178.068,7.121,148.767
C06136=1158.065,194.938,-61.100,-178.070,7.119,148.767
C06137=1158.069,194.689,-61.077,-178.073,7.117,148.768
C06138=1158.074,194.441,-61.053,-178.076,7.114,148.768
C06139=1158.078,194.192,-61.029,-178.078,7.112,148.768
C06140=1158.083,193.943,-61.005,-178.082,7.110,148.768
C06141=1158.088,193.694,-60.982,-178.084,7.108,148.768
C06142=1158.092,193.445,-60.959,-178.087,7.105,148.769
C06143=1158.097,193.197,-60.934,-178.090,7.103,148.769
C06144=1158.102,192.948,-60.910,-178.092,7.101,148.769
C06145=1158.107,192.699,-60.887,-178.095,7.098,148.770
C06146=1158.111,192.450,-60.863,-178.098,7.097,148.770
C06147=1158.116,192.201,-60.840,-178.101,7.094,148.770
C06148=1158.121,191.952,-60.816,-178.103,7.092,148.770
C06149=1158.125,191.704,-60.792,-178.106,7.090,148.771
C06150=1158.129,191.455,-60.769,-178.109,7.087,148.771
C06151=1158.134,191.206,-60.746,-178.112,7.086,148.771
C06152=1158.138,190.957,-60.723,-178.114,7.083,148.771
C06153=1158.143,190.709,-60.699,-178.117,7.081,148.772
C06154=1158.147,190.459,-60.675,-178.120,7.079,148.772
C06155=1158.152,190.210,-60.652,-178.123,7.076,148.772
C06156=1158.157,189.961,-60.629,-178.125,7.075,148.773
C06157=1158.161,189.712,-60.605,-178.129,7.072,148.773
C06158=1158.166,189.464,-60.581,-178.131,7.070,148.773
C06159=1158.171,189.215,-60.558,-178.133,7.068,148.773
C06160=1158.175,188.966,-60.534,-178.136,7.065,148.773
C06161=1158.180,188.717,-60.511,-178.139,7.063,148.774
C06162=1158.185,188.468,-60.488,-178.142,7.061,148.774
C06163=1158.189,188.219,-60.465,-178.144,7.059,148.774
C06164=1158.193,187.970,-60.442,-178.147,7.057,148.775
C06165=1158.198,187.722,-60.418,-178.150,7.054,148.775
C06166=1158.203,187.473,-60.395,-178.153,7.052,148.775
C06167=1158.208,187.224,-60.371,-178.155,7.051,148.775
C06168=1158.212,186.975,-60.348,-178.158,7.048,148.776
C06169=1158.216,186.727,-60.325,-178.161,7.046,148.776
C06170=1158.221,186.478,-60.302,-178.164,7.043,148.776
C06171=1158.226,186.228,-60.278,-178.167,7.042,148.777
C06172=1158.231,185.979,-60.255,-178.169,7.039,148.777
C06173=1158.235,185.730,-60.232,-178.172,7.037,148.777
C06174=1158.239,185.482,-60.209,-178.175,7.035,148.777
C06175=1158.244,185.233,-60.186,-178.177,7.033,148.778
C06176=1158.249,184.984,-60.163,-178.180,7.030,148.778
C06177=1158.254,184.735,-60.139,-178.183,7.029,148.778
C06178=1158.258,184.487,-60.116,-178.186,7.027,148.779
C06179=1158.263,184.217,-60.091,-178.188,7.024,148.779
C06180=1158.268,183.947,-60.066,-178.192,7.021,148.779
C06181=1158.273,183.678,-60.042,-178.194,7.020,148.780
C06182=1158.278,183.408,-60.017,-178.198,7.017,148.780
C06183=1158.283,183.159,-59.994,-178.200,7.015,148.780
C06184=1158.287,182.910,-59.971,-178.203,7.012,148.780
C06185=1158.292,182.661,-59.947,-178.206,7.011,148.781
C06186=1158.296,182.412,-59.924,-178.209,7.009,148.781
C06187=1158.301,182.164,-59.902,-178.211,7.006,148.781
C06188=1158.306,181.915,-59.878,-178.214,7.004,148.782
C06189=1158.311,181.665,-59.856,-178.217,7.003,148.782
C06190=1158.315,181.417,-59.833,-178.220,7.000,148.782
C06191=1158.319,181.168,-59.809,-178.222,6.998,148.782
C06192=1158.325,180.919,-59.787,-178.225,6.996,148.783
C06193=1158.329,180.670,-59.764,-178.228,6.994,148.783
C06194=1158.334,180.421,-59.741,-178.231,6.992,148.783
C06195=1158.338,180.172,-59.718,-178.233,6.990,148.784
C06196=1158.342,179.923,-59.695,-178.236,6.987,148.784
C06197=1158.348,179.674,-59.673,-178.239,6.985,148.784
C06198=1158.352,179.425,-59.650,-178.241,6.983,148.784
C06199=1158.357,179.176,-59.627,-178.244,6.981,148.785
C06200=1158.361,178.927,-59.605,-178.247,6.979,148.785
C06201=1158.366,178.679,-59.582,-178.250,6.977,148.785
C06202=1158.370,178.430,-59.559,-178.252,6.975,148.786
C06203=1158.375,178.180,-59.536,-178.255,6.973,148.786
C06204=1158.380,177.931,-59.513,-178.258,6.971,148.786
C06205=1158.384,177.683,-59.490,-178.261,6.969,148.787
C06206=1158.389,177.434,-59.468,-178.264,6.966,148.787
C06207=1158.393,177.185,-59.445,-178.266,6.964,148.787
C06208=1158.399,176.936,-59.423,-178.269,6.963,148.788
C06209=1158.403,176.687,-59.400,-178.272,6.960,148.788
C06210=1158.408,176.438,-59.377,-178.274,6.958,148.788
C06211=1158.412,176.190,-59.355,-178.277,6.956,148.788
C06212=1158.416,175.941,-59.332,-178.280,6.954,148.789
C06213=1158.421,175.691,-59.309,-178.283,6.952,148.789
C06214=1158.425,175.442,-59.287,-178.285,6.950,148.789
C06215=1158.431,175.194,-59.264,-178.288,6.948,148.790
C06216=1158.435,174.945,-59.242,-178.291,6.945,148.790
C06217=1158.440,174.695,-59.219,-178.294,6.944,148.790
C06218=1158.445,174.447,-59.197,-178.297,6.942,148.791
C06219=1158.450,174.197,-59.174,-178.299,6.940,148.791
C06220=1158.454,173.949,-59.152,-178.302,6.937,148.791
C06221=1158.458,173.700,-59.130,-178.305,6.936,148.792
C06222=1158.463,173.450,-59.107,-178.307,6.934,148.792
C06223=1158.468,173.202,-59.084,-178.310,6.932,148.792
C06224=1158.472,172.953,-59.062,-178.313,6.929,148.792
C06225=1158.477,172.704,-59.039,-178.316,6.927,148.793
C06226=1158.482,172.455,-59.017,-178.318,6.926,148.793
C06227=1158.487,172.206,-58.995,-178.322,6.923,148.793
C06228=1158.491,171.958,-58.972,-178.324,6.921,148.794
C06229=1158.496,171.708,-58.950,-178.327,6.919,148.794
C06230=1158.501,171.459,-58.928,-178.329,6.918,148.794
C06231=1158.505,171.211,-58.905,-178.332,6.915,148.795
C06232=1158.509,170.961,-58.883,-178.335,6.913,148.795
C06233=1158.514,170.713,-58.862,-178.337,6.911,148.795
C06234=1158.519,170.463,-58.839,-178.340,6.909,148.796
C06235=1158.524,170.215,-58.817,-178.343,6.907,148.796
C06236=1158.528,169.966,-58.794,-178.346,6.905,148.796
C06237=1158.533,169.716,-58.772,-178.349,6.903,148.797
C06238=1158.538,169.467,-58.750,-178.351,6.901,148.797
C06239=1158.542,169.219,-58.727,-178.354,6.899,148.797
C06240=1158.547,168.970,-58.706,-178.357,6.897,148.798
C06241=1158.552,168.720,-58.683,-178.360,6.895,148.798
C06242=1158.557,168.472,-58.661,-178.362,6.893,148.798
C06243=1158.561,168.222,-58.639,-178.365,6.892,148.799
C06244=1158.566,167.974,-58.617,-178.368,6.889,148.799
C06245=1158.571,167.725,-58.594,-178.371,6.887,148.799
C06246=1158.575,167.476,-58.573,-178.373,6.885,148.800
C06247=1158.580,167.227,-58.551,-178.376,6.884,148.800
C06248=1158.585,166.978,-58.529,-178.379,6.881,148.800
C06249=1158.589,166.729,-58.507,-178.382,6.879,148.801
C06250=1158.594,166.480,-58.485,-178.384,6.877,148.801
C06251=1158.599,166.231,-58.462,-178.387,6.875,148.801
C06252=1158.604,165.982,-58.441,-178.389,6.874,148.802
C06253=1158.608,165.733,-58.419,-178.393,6.871,148.802
C06254=1158.613,165.484,-58.397,-178.395,6.869,148.802
C06255=1158.617,165.235,-58.375,-178.398,6.868,148.803
C06256=1158.622,164.987,-58.353,-178.400,6.866,148.803
C06257=1158.626,164.737,-58.331,-178.404,6.863,148.803
C06258=1158.631,164.488,-58.308,-178.406,6.861,148.803
C06259=1158.636,164.238,-58.287,-178.409,6.860,148.804
C06260=1158.641,163.990,-58.265,-178.412,6.858,148.804
C06261=1158.645,163.740,-58.243,-178.414,6.856,148.805
C06262=1158.650,163.492,-58.222,-178.418,6.853,148.805
C06263=1158.655,163.243,-58.200,-178.420,6.851,148.805
C06264=1158.659,162.994,-58.178,-178.423,6.850,148.805
C06265=1158.664,162.745,-58.156,-178.425,6.848,148.806
C06266=1158.668,162.496,-58.134,-178.428,6.846,148.806
C06267=1158.673,162.247,-58.112,-178.431,6.844,148.807
C06268=1158.677,161.998,-58.090,-178.434,6.842,148.807
C06269=1158.682,161.749,-58.069,-178.437,6.840,148.807
C06270=1158.687,161.500,-58.047,-178.439,6.838,148.808
C06271=1158.692,161.250,-58.026,-178.442,6.836,148.808
C06272=1158.697,161.002,-58.004,-178.444,6.835,148.808
C06273=1158.701,160.753,-57.982,-178.448,6.832,148.809
C06274=1158.706,160.504,-57.960,-178.450,6.830,148.809
C06275=1158.711,160.255,-57.939,-178.453,6.829,148.809
C06276=1158.715,160.005,-57.917,-178.456,6.827,148.810
C06277=1158.720,159.757,-57.896,-178.458,6.825,148.810
C06278=1158.725,159.508,-57.874,-178.461,6.823,148.810
C06279=1158.729,159.259,-57.852,-178.464,6.820,148.811
C06280=1158.734,159.010,-57.830,-178.467,6.819,148.811
C06281=1158.739,158.761,-57.809,-178.469,6.817,148.811
C06282=1158.744,158.511,-57.787,-178.472,6.815,148.812
C06283=1158.748,158.242,-57.764,-178.475,6.813,148.812
C06284=1158.753,157.974,-57.740,-178.478,6.811,148.812
C06285=1158.759,157.705,-57.718,-178.481,6.809,148.813
C06286=1158.764,157.436,-57.695,-178.484,6.807,148.813
C06287=1158.769,157.187,-57.672,-178.487,6.805,148.814
C06288=1158.773,156.938,-57.652,-178.489,6.803,148.814
C06289=1158.778,156.689,-57.630,-178.492,6.801,148.814
C06290=1158.782,156.440,-57.608,-178.495,6.800,148.815
C06291=1158.787,156.190,-57.587,-178.497,6.798,148.815
C06292=1158.792,155.942,-57.566,-178.501,6.795,148.815
C06293=1158.797,155.693,-57.544,-178.503,6.794,148.816
C06294=1158.801,155.443,-57.523,-178.506,6.792,148.816
C06295=1158.806,155.195,-57.502,-178.509,6.790,148.817
C06296=1158.811,154.946,-57.481,-178.511,6.788,148.817
C06297=1158.815,154.696,-57.459,-178.514,6.786,148.817
C06298=1158.820,154.447,-57.438,-178.516,6.785,148.817
C06299=1158.825,154.198,-57.416,-178.519,6.783,148.818
C06300=1158.830,153.949,-57.396,-178.522,6.780,148.818
C06301=1158.835,153.701,-57.374,-178.525,6.779,148.819
C06302=1158.839,153.451,-57.353,-178.528,6.777,148.819
C06303=1158.844,153.202,-57.331,-178.530,6.775,148.819
C06304=1158.848,152.953,-57.311,-178.533,6.773,148.820
C06305=1158.853,152.705,-57.289,-178.536,6.772,148.820
C06306=1158.858,152.455,-57.268,-178.539,6.770,148.821
C06307=1158.863,152.206,-57.246,-178.541,6.768,148.821
C06308=1158.867,151.957,-57.225,-178.545,6.766,148.821
C06309=1158.872,151.708,-57.204,-178.547,6.764,148.822
C06310=1158.877,151.459,-57.183,-178.550,6.762,148.822
C06311=1158.881,151.209,-57.162,-178.553,6.760,148.822
C06312=1158.886,150.961,-57.140,-178.555,6.759,148.823
C06313=1158.891,150.712,-57.119,-178.558,6.757,148.823
C06314=1158.896,150.463,-57.099,-178.560,6.755,148.823
C06315=1158.900,150.214,-57.077,-178.563,6.753,148.824
C06316=1158.906,149.965,-57.056,-178.566,6.751,148.824
C06317=1158.909,149.715,-57.036,-178.568,6.750,148.824
C06318=1158.914,149.466,-57.014,-178.572,6.747,148.825
C06319=1158.919,149.217,-56.993,-178.574,6.745,148.825
C06320=1158.924,148.968,-56.973,-178.577,6.744,148.826
C06321=1158.929,148.719,-56.952,-178.580,6.742,148.826
C06322=1158.934,148.470,-56.930,-178.582,6.740,148.826
C06323=1158.938,148.221,-56.910,-178.585,6.738,148.827
C06324=1158.943,147.971,-56.888,-178.588,6.737,148.827
C06325=1158.947,147.722,-56.868,-178.591,6.735,148.828
C06326=1158.952,147.474,-56.846,-178.593,6.733,148.828
C06327=1158.957,147.225,-56.825,-178.596,6.732,148.828
C06328=1158.962,146.976,-56.805,-178.599,6.730,148.829
C06329=1158.967,146.726,-56.784,-178.601,6.728,148.829
C06330=1158.971,146.477,-56.764,-178.605,6.726,148.829
C06331=1158.977,146.228,-56.743,-178.607,6.724,148.830
C06332=1158.981,145.980,-56.721,-178.610,6.722,148.830
C06333=1158.985,145.730,-56.700,-178.613,6.720,148.831
C06334=1158.990,145.481,-56.680,-178.616,6.719,148.831
C06335=1158.995,145.232,-56.659,-178.618,6.717,148.831
C06336=1158.999,144.983,-56.638,-178.621,6.715,148.832
C06337=1159.005,144.733,-56.617,-178.624,6.713,148.832
C06338=1159.009,144.484,-56.597,-178.626,6.712,148.832
C06339=1159.014,144.235,-56.576,-178.629,6.710,148.833
C06340=1159.019,143.986,-56.556,-178.632,6.708,148.833
C06341=1159.024,143.737,-56.535,-178.634,6.706,148.834
C06342=1159.028,143.488,-56.514,-178.637,6.705,148.834
C06343=1159.033,143.239,-56.493,-178.640,6.703,148.834
C06344=1159.038,142.990,-56.472,-178.643,6.701,148.835
C06345=1159.042,142.742,-56.452,-178.645,6.700,148.835
C06346=1159.047,142.492,-56.432,-178.648,6.698,148.836
C06347=1159.052,142.243,-56.411,-178.651,6.696,148.836
C06348=1159.057,141.993,-56.390,-178.653,6.694,148.836
C06349=1159.061,141.744,-56.370,-178.656,6.693,148.837
C06350=1159.067,141.495,-56.349,-178.659,6.690,148.837
C06351=1159.071,141.246,-56.329,-178.662,6.688,148.837
C06352=1159.076,140.997,-56.308,-178.665,6.687,148.838
C06353=1159.081,140.748,-56.287,-178.667,6.685,148.838
C06354=1159.085,140.499,-56.267,-178.670,6.683,148.839
C06355=1159.090,140.250,-56.247,-178.673,6.681,148.839
C06356=1159.095,140.001,-56.226,-178.676,6.680,148.839
C06357=1159.099,139.752,-56.205,-178.678,6.678,148.840
C06358=1159.104,139.503,-56.185,-178.681,6.676,148.840
C06359=1159.109,139.253,-56.165,-178.684,6.675,148.841
C06360=1159.114,139.004,-56.144,-178.686,6.673,148.841
C06361=1159.118,138.755,-56.124,-178.689,6.671,148.841
C06362=1159.123,138.506,-56.103,-178.692,6.669,148.842
C06363=1159.128,138.257,-56.083,-178.695,6.668,148.842
C06364=1159.132,138.007,-56.063,-178.698,6.666,148.843
C06365=1159.138,137.758,-56.042,-178.700,6.665,148.843
C06366=1159.142,137.509,-56.022,-178.703,6.663,148.844
C06367=1159.146,137.260,-56.001,-178.706,6.661,148.844
C06368=1159.151,137.011,-55.981,-178.709,6.659,148.844
C06369=1159.156,136.761,-55.961,-178.711,6.658,148.845
C06370=1159.161,136.513,-55.941,-178.714,6.656,148.845
C06371=1159.166,136.264,-55.920,-178.717,6.654,148.845
C06372=1159.171,136.015,-55.901,-178.719,6.652,148.846
C06373=1159.176,135.765,-55.880,-178.722,6.651,148.846
C06374=1159.180,135.516,-55.859,-178.725,6.649,148.847
C06375=1159.185,135.267,-55.840,-178.728,6.647,148.847
C06376=1159.189,135.018,-55.819,-178.730,6.646,148.847
C06377=1159.194,134.769,-55.799,-178.733,6.644,148.848
C06378=1159.200,134.520,-55.779,-178.736,6.642,148.848
C06379=1159.204,134.271,-55.759,-178.738,6.640,148.849
C06380=1159.209,134.022,-55.738,-178.741,6.639,148.849
C06381=1159.213,133.772,-55.719,-178.744,6.637,148.850
C06382=1159.218,133.523,-55.698,-178.747,6.636,148.850
C06383=1159.223,133.274,-55.679,-178.750,6.634,148.850
C06384=1159.228,133.025,-55.658,-178.752,6.632,148.851
C06385=1159.233,132.776,-55.638,-178.755,6.630,148.851
C06386=1159.238,132.527,-55.618,-178.758,6.629,148.852
C06387=1159.243,132.258,-55.597,-178.761,6.627,148.852
C06388=1159.248,131.990,-55.574,-178.763,6.625,148.852
C06389=1159.253,131.721,-55.553,-178.766,6.624,148.853
C06390=1159.258,131.452,-55.532,-178.769,6.622,148.853
C06391=1159.263,131.203,-55.511,-178.772,6.620,148.854
C06392=1159.268,130.954,-55.492,-178.775,6.619,148.854
C06393=1159.272,130.705,-55.471,-178.777,6.617,148.855
C06394=1159.277,130.456,-55.452,-178.780,6.615,148.855
C06395=1159.282,130.207,-55.432,-178.783,6.614,148.855
C06396=1159.287,129.957,-55.412,-178.785,6.612,148.856
C06397=1159.291,129.708,-55.392,-178.789,6.611,148.856
C06398=1159.296,129.460,-55.372,-178.791,6.609,148.857
C06399=1159.301,129.210,-55.353,-178.794,6.607,148.857
C06400=1159.306,128.961,-55.332,-178.797,6.605,148.858
C06401=1159.310,128.711,-55.313,-178.799,6.604,148.858
C06402=1159.315,128.463,-55.293,-178.802,6.602,148.858
C06403=1159.320,128.214,-55.273,-178.805,6.600,148.859
C06404=1159.325,127.964,-55.253,-178.808,6.598,148.859
C06405=1159.329,127.715,-55.233,-178.810,6.598,148.860
C06406=1159.335,127.466,-55.214,-178.812,6.596,148.860
C06407=1159.339,127.217,-55.194,-178.816,6.594,148.861
C06408=1159.344,126.968,-55.174,-178.818,6.593,148.861
C06409=1159.349,126.718,-55.154,-178.821,6.591,148.861
C06410=1159.354,126.469,-55.135,-178.824,6.589,148.862
C06411=1159.359,126.220,-55.115,-178.826,6.588,148.862
C06412=1159.363,125.971,-55.095,-178.829,6.586,148.863
C06413=1159.368,125.722,-55.075,-178.832,6.584,148.863
C06414=1159.373,125.472,-55.056,-178.835,6.582,148.863
C06415=1159.378,125.223,-55.036,-178.838,6.581,148.864
C06416=1159.382,124.974,-55.016,-178.840,6.579,148.864
C06417=1159.387,124.725,-54.997,-178.843,6.578,148.865
C06418=1159.392,124.476,-54.977,-178.845,6.577,148.865
C06419=1159.396,124.226,-54.958,-178.848,6.575,148.866
C06420=1159.402,123.977,-54.938,-178.851,6.573,148.866
C06421=1159.406,123.728,-54.919,-178.853,6.572,148.866
C06422=1159.411,123.479,-54.898,-178.856,6.570,148.867
C06423=1159.416,123.230,-54.880,-178.859,6.569,148.867
C06424=1159.420,122.981,-54.860,-178.862,6.567,148.868
C06425=1159.426,122.732,-54.841,-178.865,6.565,148.868
C06426=1159.430,122.482,-54.821,-178.868,6.563,148.869
C06427=1159.435,122.233,-54.801,-178.870,6.562,148.869
C06428=1159.440,121.984,-54.782,-178.872,6.561,148.869
C06429=1159.444,121.734,-54.763,-178.875,6.559,148.870
C06430=1159.449,121.485,-54.743,-178.878,6.558,148.870
C06431=1159.454,121.237,-54.723,-178.881,6.556,148.871
C06432=1159.459,120.987,-54.704,-178.884,6.554,148.871
C06433=1159.464,120.738,-54.684,-178.886,6.553,148.872
C06434=1159.468,120.489,-54.665,-178.889,6.551,148.872
C06435=1159.473,120.239,-54.646,-178.892,6.549,148.872
C06436=1159.478,119.991,-54.626,-178.894,6.549,148.873
C06437=1159.483,119.741,-54.607,-178.897,6.547,148.873
C06438=1159.488,119.492,-54.588,-178.900,6.545,148.874
C06439=1159.492,119.243,-54.568,-178.903,6.543,148.874
C06440=1159.497,118.993,-54.549,-178.905,6.542,148.875
C06441=1159.503,118.744,-54.529,-178.908,6.540,148.875
C06442=1159.507,118.495,-54.511,-178.911,6.538,148.875
C06443=1159.512,118.246,-54.492,-178.914,6.537,148.876
C06444=1159.517,117.996,-54.472,-178.916,6.536,148.876
C06445=1159.522,117.748,-54.453,-178.919,6.534,148.877
C06446=1159.526,117.498,-54.434,-178.922,6.533,148.877
C06447=1159.532,117.249,-54.414,-178.924,6.531,148.878
C06448=1159.536,117.000,-54.395,-178.927,6.530,148.878
C06449=1159.541,116.751,-54.376,-178.930,6.528,148.879
C06450=1159.546,116.501,-54.356,-178.933,6.526,148.879
C06451=1159.550,116.252,-54.338,-178.935,6.525,148.880
C06452=1159.555,116.003,-54.319,-178.938,6.524,148.880
C06453=1159.560,115.753,-54.299,-178.940,6.522,148.880
C06454=1159.565,115.505,-54.280,-178.944,6.520,148.881
C06455=1159.570,115.255,-54.261,-178.946,6.519,148.881
C06456=1159.574,115.006,-54.243,-178.949,6.517,148.882
C06457=1159.579,114.756,-54.223,-178.951,6.516,148.882
C06458=1159.585,114.507,-54.204,-178.954,6.514,148.883
C06459=1159.589,114.259,-54.185,-178.957,6.513,148.883
C06460=1159.594,114.009,-54.166,-178.960,6.511,148.884
C06461=1159.599,113.760,-54.148,-178.963,6.510,148.884
C06462=1159.604,113.510,-54.128,-178.965,6.508,148.884
C06463=1159.609,113.262,-54.109,-178.967,6.507,148.885
C06464=1159.613,113.012,-54.090,-178.970,6.505,148.885
C06465=1159.619,112.763,-54.071,-178.973,6.504,148.886
C06466=1159.623,112.514,-54.052,-178.976,6.502,148.886
C06467=1159.628,112.264,-54.033,-178.979,6.501,148.887
C06468=1159.632,112.015,-54.014,-178.981,6.499,148.887
C06469=1159.638,111.766,-53.995,-178.984,6.498,148.888
C06470=1159.642,111.517,-53.977,-178.987,6.497,148.888
C06471=1159.647,111.267,-53.957,-178.990,6.495,148.889
C06472=1159.652,111.019,-53.939,-178.992,6.493,148.889
C06473=1159.657,110.769,-53.920,-178.995,6.492,148.889
C06474=1159.661,110.520,-53.901,-178.998,6.491,148.890
C06475=1159.667,110.270,-53.882,-179.000,6.489,148.890
C06476=1159.671,110.021,-53.863,-179.003,6.488,148.891
C06477=1159.676,109.772,-53.844,-179.006,6.486,148.891
C06478=1159.681,109.522,-53.826,-179.008,6.484,148.892
C06479=1159.686,109.274,-53.806,-179.011,6.484,148.892
C06480=1159.691,109.024,-53.788,-179.014,6.482,148.893
C06481=1159.695,108.775,-53.769,-179.017,6.480,148.893
C06482=1159.701,108.526,-53.751,-179.019,6.479,148.893
C06483=1159.705,108.276,-53.732,-179.022,6.477,148.894
C06484=1159.710,108.027,-53.713,-179.025,6.476,148.895
C06485=1159.715,107.778,-53.695,-179.027,6.475,148.895
C06486=1159.719,107.529,-53.676,-179.030,6.473,148.895
C06487=1159.725,107.280,-53.657,-179.033,6.471,148.896
C06488=1159.729,107.030,-53.639,-179.036,6.470,148.896
C06489=1159.735,106.780,-53.620,-179.038,6.469,148.897
C06490=1159.739,106.532,-53.601,-179.041,6.467,148.897
C06491=1159.744,106.263,-53.582,-179.044,6.466,148.898
C06492=1159.749,105.995,-53.561,-179.047,6.464,148.898
C06493=1159.754,105.727,-53.541,-179.049,6.462,148.899
C06494=1159.760,105.458,-53.521,-179.053,6.461,148.899
C06495=1159.765,105.209,-53.503,-179.055,6.459,148.900
C06496=1159.770,104.959,-53.484,-179.058,6.458,148.900
C06497=1159.775,104.710,-53.466,-179.060,6.457,148.901
C06498=1159.779,104.462,-53.447,-179.063,6.455,148.901
C06499=1159.784,104.212,-53.429,-179.066,6.454,148.902
C06500=1159.789,103.962,-53.410,-179.069,6.452,148.902
C06501=1159.794,103.714,-53.391,-179.071,6.451,148.902
C06502=1159.799,103.464,-53.373,-179.074,6.450,148.903
C06503=1159.804,103.214,-53.354,-179.077,6.448,148.903
C06504=1159.809,102.965,-53.337,-179.080,6.446,148.904
C06505=1159.813,102.717,-53.318,-179.082,6.446,148.904
C06506=1159.818,102.467,-53.300,-179.085,6.444,148.905
C06507=1159.823,102.217,-53.281,-179.088,6.443,148.905
C06508=1159.828,101.968,-53.263,-179.090,6.441,148.906
C06509=1159.833,101.719,-53.244,-179.093,6.440,148.906
C06510=1159.838,101.470,-53.226,-179.096,6.439,148.907
C06511=1159.843,101.220,-53.207,-179.099,6.437,148.907
C06512=1159.848,100.971,-53.189,-179.101,6.435,148.908
C06513=1159.853,100.722,-53.171,-179.104,6.435,148.908
C06514=1159.857,100.473,-53.153,-179.107,6.433,148.909
C06515=1159.861,100.223,-53.134,-179.109,6.431,148.909
C06516=1159.866,99.974,-53.116,-179.112,6.430,148.910
C06517=1159.872,99.725,-53.098,-179.115,6.429,148.910
C06518=1159.877,99.475,-53.080,-179.117,6.427,148.911
C06519=1159.882,99.226,-53.062,-179.120,6.426,148.911
C06520=1159.886,98.976,-53.043,-179.123,6.424,148.911
C06521=1159.891,98.728,-53.025,-179.125,6.423,148.912
C06522=1159.896,98.479,-53.007,-179.128,6.422,148.912
C06523=1159.901,98.229,-52.989,-179.131,6.420,148.913
C06524=1159.906,97.980,-52.970,-179.133,6.419,148.913
C06525=1159.911,97.731,-52.952,-179.136,6.418,148.914
C06526=1159.915,97.481,-52.934,-179.139,6.416,148.914
C06527=1159.920,97.232,-52.916,-179.142,6.414,148.915
C06528=1159.925,96.983,-52.898,-179.144,6.414,148.915
C06529=1159.930,96.733,-52.880,-179.147,6.412,148.916
C06530=1159.935,96.484,-52.862,-179.150,6.410,148.916
C06531=1159.940,96.235,-52.844,-179.152,6.410,148.917
C06532=1159.944,95.985,-52.826,-179.155,6.408,148.917
C06533=1159.949,95.736,-52.808,-179.158,6.407,148.918
C06534=1159.954,95.487,-52.790,-179.161,6.405,148.918
C06535=1159.959,95.238,-52.772,-179.163,6.404,148.919
C06536=1159.964,94.988,-52.754,-179.166,6.403,148.919
C06537=1159.969,94.739,-52.736,-179.169,6.401,148.920
C06538=1159.975,94.490,-52.717,-179.171,6.400,148.920
C06539=1159.979,94.241,-52.699,-179.174,6.399,148.921
C06540=1159.984,93.991,-52.681,-179.177,6.397,148.921
C06541=1159.989,93.742,-52.663,-179.179,6.396,148.922
C06542=1159.994,93.492,-52.646,-179.182,6.395,148.922
C06543=1159.999,93.243,-52.628,-179.185,6.393,148.923
C06544=1160.003,92.994,-52.610,-179.187,6.392,148.923
C06545=1160.008,92.745,-52.592,-179.190,6.391,148.924
C06546=1160.013,92.495,-52.574,-179.193,6.389,148.924
C06547=1160.018,92.246,-52.556,-179.196,6.387,148.924
C06548=1160.023,91.997,-52.538,-179.198,6.387,148.925
C06549=1160.028,91.747,-52.521,-179.201,6.385,148.926
C06550=1160.033,91.498,-52.503,-179.204,6.384,148.926
C06551=1160.038,91.249,-52.485,-179.206,6.383,148.926
C06552=1160.043,91.000,-52.467,-179.209,6.381,148.927
C06553=1160.047,90.751,-52.449,-179.212,6.380,148.927
C06554=1160.052,90.500,-52.431,-179.214,6.379,148.928
C06555=1160.057,90.251,-52.414,-179.217,6.377,148.929
C06556=1160.062,90.002,-52.396,-179.220,6.376,148.929
C06557=1160.067,89.753,-52.378,-179.222,6.375,148.929
C06558=1160.071,89.503,-52.361,-179.225,6.374,148.930
C06559=1160.076,89.254,-52.343,-179.228,6.372,148.930
C06560=1160.081,89.005,-52.325,-179.230,6.371,148.931
C06561=1160.086,88.755,-52.308,-179.233,6.370,148.931
C06562=1160.091,88.506,-52.290,-179.236,6.368,148.932
C06563=1160.096,88.257,-52.272,-179.238,6.367,148.932
C06564=1160.101,88.007,-52.254,-179.241,6.366,148.933
C06565=1160.106,87.758,-52.237,-179.243,6.365,148.933
C06566=1160.110,87.509,-52.219,-179.246,6.363,148.934
C06567=1160.116,87.259,-52.202,-179.249,6.362,148.934
C06568=1160.121,87.010,-52.184,-179.252,6.361,148.935
C06569=1160.126,86.761,-52.166,-179.254,6.359,148.935
C06570=1160.130,86.511,-52.149,-179.258,6.358,148.936
C06571=1160.135,86.263,-52.132,-179.260,6.357,148.936
C06572=1160.141,86.013,-52.114,-179.262,6.355,148.937
C06573=1160.146,85.764,-52.096,-179.266,6.354,148.937
C06574=1160.151,85.514,-52.079,-179.268,6.353,148.938
C06575=1160.155,85.265,-52.062,-179.270,6.351,148.938
C06576=1160.160,85.016,-52.044,-179.273,6.351,148.939
C06577=1160.165,84.766,-52.026,-179.276,6.349,148.939
C06578=1160.170,84.517,-52.008,-179.279,6.348,148.940
C06579=1160.175,84.267,-51.992,-179.281,6.347,148.940
C06580=1160.179,84.018,-51.974,-179.284,6.345,148.941
C06581=1160.185,83.768,-51.957,-179.287,6.344,148.941
C06582=1160.189,83.520,-51.939,-179.289,6.343,148.942
C06583=1160.194,83.270,-51.922,-179.292,6.341,148.942
C06584=1160.199,83.021,-51.904,-179.294,6.341,148.943
C06585=1160.204,82.771,-51.887,-179.297,6.339,148.943
C06586=1160.209,82.522,-51.870,-179.300,6.338,148.944
C06587=1160.214,82.273,-51.852,-179.302,6.337,148.944
C06588=1160.219,82.023,-51.835,-179.305,6.335,148.945
C06589=1160.224,81.774,-51.818,-179.308,6.334,148.945
C06590=1160.229,81.524,-51.800,-179.310,6.333,148.946
C06591=1160.234,81.275,-51.782,-179.314,6.332,148.946
C06592=1160.238,81.026,-51.766,-179.316,6.331,148.947
C06593=1160.243,80.776,-51.749,-179.319,6.329,148.948
C06594=1160.248,80.528,-51.732,-179.322,6.328,148.948
C06595=1160.254,80.259,-51.713,-179.324,6.327,148.948
C06596=1160.259,79.990,-51.694,-179.327,6.325,148.949
C06597=1160.264,79.722,-51.676,-179.330,6.324,148.950
C06598=1160.269,79.454,-51.657,-179.333,6.322,148.950
C06599=1160.275,79.204,-51.640,-179.335,6.322,148.951
C06600=1160.279,78.955,-51.623,-179.338,6.320,148.951
C06601=1160.284,78.705,-51.606,-179.340,6.319,148.952
C06602=1160.290,78.456,-51.588,-179.344,6.318,148.952
C06603=1160.294,78.207,-51.572,-179.346,6.316,148.953
C06604=1160.299,77.957,-51.554,-179.349,6.315,148.953
C06605=1160.304,77.708,-51.538,-179.352,6.314,148.954
C06606=1160.309,77.458,-51.520,-179.354,6.313,148.954
C06607=1160.314,77.210,-51.503,-179.357,6.312,148.955
C06608=1160.319,76.960,-51.486,-179.360,6.310,148.955
C06609=1160.324,76.710,-51.469,-179.362,6.309,148.956
C06610=1160.329,76.461,-51.451,-179.365,6.308,148.956
C06611=1160.333,76.212,-51.435,-179.367,6.307,148.957
C06612=1160.339,75.963,-51.418,-179.370,6.306,148.957
C06613=1160.343,75.713,-51.401,-179.373,6.305,148.958
C06614=1160.349,75.463,-51.384,-179.375,6.303,148.958
C06615=1160.353,75.214,-51.367,-179.378,6.302,148.959
C06616=1160.358,74.965,-51.350,-179.381,6.301,148.959
C06617=1160.363,74.716,-51.333,-179.384,6.299,148.960
C06618=1160.368,74.466,-51.316,-179.386,6.299,148.960
C06619=1160.373,74.217,-51.299,-179.389,6.297,148.961
C06620=1160.378,73.967,-51.282,-179.391,6.296,148.961
C06621=1160.383,73.718,-51.265,-179.394,6.295,148.962
C06622=1160.388,73.468,-51.248,-179.396,6.294,148.962
C06623=1160.393,73.219,-51.231,-179.399,6.293,148.963
C06624=1160.398,72.970,-51.215,-179.402,6.292,148.964
C06625=1160.403,72.720,-51.198,-179.405,6.290,148.964
C06626=1160.407,72.471,-51.181,-179.408,6.289,148.965
C06627=1160.413,72.222,-51.164,-179.410,6.288,148.965
C06628=1160.417,71.973,-51.147,-179.413,6.286,148.965
C06629=1160.422,71.723,-51.130,-179.415,6.286,148.966
C06630=1160.427,71.473,-51.113,-179.418,6.284,148.967
C06631=1160.432,71.225,-51.097,-179.421,6.284,148.967
C06632=1160.437,70.975,-51.079,-179.423,6.282,148.968
C06633=1160.442,70.725,-51.063,-179.426,6.281,148.968
C06634=1160.447,70.477,-51.046,-179.429,6.280,148.969
C06635=1160.453,70.226,-51.030,-179.431,6.279,148.969
C06636=1160.457,69.977,-51.013,-179.434,6.278,148.970
C06637=1160.462,69.728,-50.997,-179.436,6.277,148.970
C06638=1160.467,69.478,-50.980,-179.439,6.275,148.971
C06639=1160.472,69.229,-50.963,-179.442,6.275,148.971
C06640=1160.477,68.980,-50.947,-179.444,6.273,148.972
C06641=1160.482,68.730,-50.929,-179.447,6.272,148.972
C06642=1160.487,68.481,-50.913,-179.450,6.271,148.973
C06643=1160.492,68.232,-50.897,-179.453,6.269,148.973
C06644=1160.496,67.982,-50.880,-179.455,6.269,148.974
C06645=1160.502,67.733,-50.863,-179.458,6.267,148.974
C06646=1160.507,67.483,-50.847,-179.461,6.266,148.975
C06647=1160.511,67.234,-50.830,-179.463,6.265,148.975
C06648=1160.516,66.985,-50.814,-179.465,6.264,148.976
C06649=1160.522,66.735,-50.797,-179.469,6.263,148.977
C06650=1160.526,66.486,-50.780,-179.471,6.262,148.977
C06651=1160.531,66.236,-50.764,-179.474,6.260,148.978
C06652=1160.536,65.987,-50.748,-179.476,6.260,148.978
C06653=1160.542,65.738,-50.731,-179.479,6.258,148.979
C06654=1160.546,65.488,-50.714,-179.482,6.257,148.979
C06655=1160.551,65.239,-50.698,-179.484,6.256,148.980
C06656=1160.556,64.989,-50.682,-179.487,6.255,148.980
C06657=1160.560,64.740,-50.665,-179.490,6.254,148.981
C06658=1160.566,64.491,-50.648,-179.492,6.253,148.981
C06659=1160.571,64.241,-50.632,-179.495,6.251,148.982
C06660=1160.576,63.992,-50.616,-179.498,6.251,148.982
C06661=1160.581,63.742,-50.599,-179.500,6.250,148.983
C06662=1160.585,63.493,-50.583,-179.503,6.248,148.983
C06663=1160.591,63.243,-50.567,-179.505,6.248,148.984
C06664=1160.596,62.994,-50.550,-179.508,6.246,148.984
C06665=1160.601,62.745,-50.534,-179.511,6.246,148.985
C06666=1160.606,62.495,-50.518,-179.513,6.244,148.986
C06667=1160.611,62.246,-50.501,-179.516,6.243,148.986
C06668=1160.615,61.996,-50.485,-179.519,6.242,148.987
C06669=1160.621,61.747,-50.469,-179.521,6.241,148.987
C06670=1160.625,61.497,-50.452,-179.524,6.240,148.988
C06671=1160.630,61.249,-50.436,-179.526,6.239,148.988
C06672=1160.636,60.998,-50.420,-179.529,6.237,148.989
C06673=1160.641,60.750,-50.403,-179.532,6.237,148.989
C06674=1160.646,60.499,-50.387,-179.535,6.235,148.990
C06675=1160.651,60.251,-50.371,-179.537,6.234,148.990
C06676=1160.655,60.001,-50.355,-179.540,6.233,148.991
C06677=1160.660,59.752,-50.339,-179.542,6.232,148.991
C06678=1160.665,59.502,-50.322,-179.544,6.231,148.992
C06679=1160.670,59.253,-50.307,-179.548,6.230,148.993
C06680=1160.675,59.003,-50.290,-179.550,6.229,148.993
C06681=1160.680,58.754,-50.274,-179.553,6.228,148.994
C06682=1160.685,58.504,-50.258,-179.555,6.227,148.994
C06683=1160.690,58.255,-50.242,-179.558,6.225,148.995
C06684=1160.695,58.006,-50.225,-179.561,6.225,148.995
C06685=1160.700,57.756,-50.210,-179.563,6.223,148.996
C06686=1160.705,57.506,-50.194,-179.566,6.223,148.996
C06687=1160.710,57.257,-50.178,-179.569,6.221,148.997
C06688=1160.715,57.008,-50.162,-179.571,6.221,148.997
C06689=1160.720,56.758,-50.145,-179.574,6.220,148.998
C06690=1160.725,56.509,-50.130,-179.577,6.218,148.999
C06691=1160.730,56.260,-50.113,-179.579,6.218,148.999
C06692=1160.735,56.010,-50.097,-179.582,6.216,149.000
C06693=1160.740,55.760,-50.081,-179.584,6.215,149.000
C06694=1160.745,55.511,-50.065,-179.587,6.214,149.001
C06695=1160.750,55.262,-50.050,-179.590,6.213,149.001
C06696=1160.755,55.012,-50.033,-179.592,6.212,149.002
C06697=1160.760,54.763,-50.017,-179.595,6.211,149.002
C06698=1160.765,54.513,-50.001,-179.597,6.210,149.003
C06699=1160.770,54.244,-49.984,-179.600,6.209,149.003
C06700=1160.776,53.976,-49.967,-179.603,6.208,149.004
C06701=1160.781,53.708,-49.950,-179.606,6.207,149.005
C06702=1160.786,53.439,-49.932,-179.609,6.205,149.005
C06703=1160.792,53.189,-49.917,-179.611,6.205,149.006
C06704=1160.797,52.940,-49.901,-179.614,6.204,149.006
C06705=1160.801,52.690,-49.886,-179.617,6.202,149.007
C06706=1160.806,52.441,-49.869,-179.619,6.202,149.007
C06707=1160.811,52.192,-49.854,-179.622,6.200,149.008
C06708=1160.816,51.942,-49.838,-179.625,6.200,149.008
C06709=1160.821,51.693,-49.822,-179.627,6.198,149.009
C06710=1160.827,51.444,-49.806,-179.629,6.197,149.009
C06711=1160.831,51.194,-49.790,-179.632,6.197,149.010
C06712=1160.836,50.945,-49.775,-179.635,6.195,149.010
C06713=1160.842,50.695,-49.759,-179.638,6.195,149.011
C06714=1160.846,50.446,-49.743,-179.640,6.193,149.012
C06715=1160.851,50.196,-49.727,-179.643,6.192,149.012
C06716=1160.857,49.947,-49.712,-179.645,6.192,149.013
C06717=1160.861,49.697,-49.696,-179.648,6.190,149.013
C06718=1160.866,49.448,-49.681,-179.650,6.189,149.014
C06719=1160.872,49.198,-49.665,-179.653,6.189,149.014
C06720=1160.876,48.949,-49.648,-179.656,6.187,149.015
C06721=1160.881,48.699,-49.633,-179.658,6.187,149.016
C06722=1160.886,48.450,-49.618,-179.661,6.185,149.016
C06723=1160.891,48.200,-49.602,-179.664,6.185,149.017
C06724=1160.896,47.951,-49.586,-179.666,6.184,149.017
C06725=1160.902,47.701,-49.571,-179.669,6.183,149.018
C06726=1160.906,47.452,-49.556,-179.671,6.182,149.018
C06727=1160.911,47.202,-49.540,-179.674,6.180,149.019
C06728=1160.916,46.953,-49.524,-179.677,6.179,149.019
C06729=1160.922,46.703,-49.509,-179.679,6.179,149.020
C06730=1160.926,46.455,-49.493,-179.682,6.177,149.020
C06731=1160.931,46.205,-49.477,-179.684,6.176,149.021
C06732=1160.936,45.955,-49.461,-179.687,6.176,149.022
C06733=1160.941,45.706,-49.446,-179.690,6.174,149.022
C06734=1160.946,45.457,-49.431,-179.692,6.174,149.023
C06735=1160.951,45.207,-49.415,-179.695,6.173,149.023
C06736=1160.956,44.958,-49.400,-179.698,6.172,149.024
C06737=1160.961,44.708,-49.384,-179.700,6.171,149.024
C06738=1160.967,44.459,-49.369,-179.703,6.170,149.025
C06739=1160.971,44.209,-49.353,-179.705,6.169,149.025
C06740=1160.976,43.960,-49.338,-179.708,6.168,149.026
C06741=1160.982,43.710,-49.323,-179.711,6.167,149.027
C06742=1160.986,43.461,-49.308,-179.713,6.166,149.027
C06743=1160.992,43.211,-49.292,-179.715,6.165,149.028
C06744=1160.997,42.961,-49.276,-179.719,6.164,149.028
C06745=1161.001,42.712,-49.261,-179.721,6.163,149.029
C06746=1161.007,42.463,-49.246,-179.724,6.163,149.029
C06747=1161.011,42.214,-49.231,-179.726,6.161,149.030
C06748=1161.017,41.964,-49.215,-179.729,6.160,149.031
C06749=1161.021,41.714,-49.199,-179.731,6.160,149.031
C06750=1161.026,41.465,-49.184,-179.734,6.158,149.032
C06751=1161.032,41.215,-49.169,-179.736,6.157,149.032
C06752=1161.036,40.966,-49.154,-179.739,6.157,149.033
C06753=1161.042,40.716,-49.139,-179.742,6.155,149.033
C06754=1161.047,40.467,-49.123,-179.744,6.155,149.034
C06755=1161.051,40.217,-49.108,-179.747,6.154,149.034
C06756=1161.057,39.968,-49.092,-179.750,6.153,149.035
C06757=1161.062,39.718,-49.078,-179.752,6.152,149.035
C06758=1161.067,39.469,-49.062,-179.755,6.151,149.036
C06759=1161.072,39.220,-49.047,-179.757,6.150,149.037
C06760=1161.077,38.970,-49.032,-179.760,6.149,149.037
C06761=1161.082,38.721,-49.017,-179.762,6.148,149.038
C06762=1161.087,38.471,-49.002,-179.765,6.147,149.038
C06763=1161.091,38.221,-48.986,-179.768,6.146,149.039
C06764=1161.097,37.972,-48.971,-179.770,6.146,149.039
C06765=1161.102,37.722,-48.957,-179.773,6.144,149.040
C06766=1161.107,37.473,-48.941,-179.776,6.144,149.041
C06767=1161.112,37.224,-48.926,-179.778,6.143,149.041
C06768=1161.117,36.974,-48.910,-179.781,6.142,149.042
C06769=1161.122,36.725,-48.896,-179.783,6.141,149.042
C06770=1161.128,36.475,-48.881,-179.786,6.140,149.043
C06771=1161.132,36.226,-48.866,-179.788,6.139,149.043
C06772=1161.138,35.976,-48.851,-179.791,6.138,149.044
C06773=1161.142,35.726,-48.835,-179.793,6.137,149.044
C06774=1161.147,35.477,-48.820,-179.796,6.137,149.045
C06775=1161.152,35.227,-48.805,-179.799,6.135,149.046
C06776=1161.157,34.978,-48.790,-179.801,6.135,149.046
C06777=1161.163,34.728,-48.776,-179.804,6.134,149.047
C06778=1161.167,34.479,-48.761,-179.807,6.132,149.047
C06779=1161.173,34.230,-48.745,-179.809,6.132,149.048
C06780=1161.178,33.980,-48.731,-179.812,6.131,149.048
C06781=1161.182,33.731,-48.716,-179.814,6.130,149.049
C06782=1161.188,33.481,-48.701,-179.817,6.129,149.050
C06783=1161.193,33.232,-48.686,-179.819,6.128,149.050
C06784=1161.198,32.982,-48.671,-179.822,6.128,149.051
C06785=1161.203,32.733,-48.656,-179.825,6.126,149.051
C06786=1161.208,32.483,-48.641,-179.827,6.126,149.052
C06787=1161.213,32.233,-48.626,-179.829,6.125,149.052
C06788=1161.218,31.984,-48.611,-179.832,6.124,149.053
C06789=1161.223,31.735,-48.597,-179.835,6.123,149.053
C06790=1161.228,31.485,-48.581,-179.837,6.122,149.054
C06791=1161.233,31.236,-48.567,-179.840,6.121,149.055
C06792=1161.238,30.986,-48.552,-179.843,6.120,149.055
C06793=1161.244,30.736,-48.537,-179.845,6.119,149.056
C06794=1161.248,30.487,-48.522,-179.848,6.119,149.056
C06795=1161.253,30.238,-48.508,-179.850,6.118,149.057
C06796=1161.258,29.988,-48.494,-179.853,6.117,149.057
C06797=1161.263,29.738,-48.478,-179.855,6.116,149.058
C06798=1161.268,29.489,-48.464,-179.858,6.115,149.059
C06799=1161.273,29.240,-48.449,-179.860,6.114,149.059
C06800=1161.279,28.990,-48.434,-179.863,6.113,149.060
C06801=1161.283,28.741,-48.419,-179.865,6.112,149.060
C06802=1161.288,28.491,-48.405,-179.868,6.112,149.061
C06803=1161.294,28.222,-48.389,-179.871,6.111,149.062
C06804=1161.299,27.953,-48.373,-179.874,6.110,149.062
C06805=1161.304,27.684,-48.357,-179.876,6.109,149.063
C06806=1161.310,27.415,-48.341,-179.879,6.108,149.063
C06807=1161.315,27.165,-48.326,-179.882,6.107,149.064
C06808=1161.321,26.916,-48.312,-179.884,6.107,149.065
C06809=1161.326,26.667,-48.297,-179.887,6.105,149.065
C06810=1161.330,26.418,-48.283,-179.890,6.105,149.066
C06811=1161.336,26.168,-48.268,-179.892,6.104,149.066
C06812=1161.341,25.918,-48.254,-179.894,6.103,149.067
C06813=1161.346,25.669,-48.239,-179.898,6.102,149.067
C06814=1161.351,25.419,-48.225,-179.900,6.101,149.068
C06815=1161.356,25.169,-48.210,-179.902,6.101,149.069
C06816=1161.360,24.920,-48.195,-179.905,6.100,149.069
C06817=1161.366,24.670,-48.181,-179.908,6.099,149.070
C06818=1161.371,24.420,-48.166,-179.910,6.098,149.070
C06819=1161.377,24.171,-48.152,-179.913,6.097,149.071
C06820=1161.381,23.922,-48.137,-179.915,6.096,149.071
C06821=1161.386,23.673,-48.123,-179.918,6.096,149.072
C06822=1161.391,23.423,-48.109,-179.920,6.094,149.072
C06823=1161.396,23.173,-48.095,-179.923,6.094,149.073
C06824=1161.402,22.923,-48.080,-179.925,6.093,149.074
C06825=1161.406,22.674,-48.065,-179.928,6.092,149.074
C06826=1161.412,22.425,-48.051,-179.930,6.091,149.075
C06827=1161.417,22.175,-48.037,-179.933,6.090,149.075
C06828=1161.422,21.926,-48.022,-179.935,6.090,149.076
C06829=1161.427,21.676,-48.008,-179.938,6.089,149.077
C06830=1161.432,21.426,-47.994,-179.941,6.089,149.077
C06831=1161.437,21.177,-47.979,-179.943,6.087,149.078
C06832=1161.441,20.927,-47.964,-179.946,6.086,149.078
C06833=1161.447,20.678,-47.951,-179.948,6.086,149.079
C06834=1161.452,20.429,-47.936,-179.951,6.085,149.079
C06835=1161.457,20.179,-47.922,-179.953,6.084,149.080
C06836=1161.462,19.929,-47.908,-179.956,6.083,149.081
C06837=1161.467,19.679,-47.893,-179.958,6.082,149.081
C06838=1161.473,19.430,-47.879,-179.961,6.082,149.082
C06839=1161.478,19.181,-47.865,-179.963,6.081,149.082
C06840=1161.483,18.931,-47.850,-179.966,6.080,149.083
C06841=1161.488,18.681,-47.836,-179.969,6.079,149.083
C06842=1161.493,18.431,-47.822,-179.971,6.078,149.084
C06843=1161.498,18.182,-47.808,-179.973,6.078,149.084
C06844=1161.503,17.933,-47.794,-179.976,6.077,149.085
C06845=1161.508,17.683,-47.779,-179.979,6.077,149.086
C06846=1161.513,17.433,-47.765,-179.981,6.075,149.086
C06847=1161.519,17.184,-47.751,-179.984,6.074,149.087
C06848=1161.524,16.935,-47.737,-179.986,6.074,149.087
C06849=1161.528,16.685,-47.723,-179.989,6.073,149.088
C06850=1161.533,16.435,-47.709,-179.991,6.072,149.089
C06851=1161.538,16.186,-47.695,-179.994,6.071,149.089
C06852=1161.543,15.937,-47.681,-179.997,6.070,149.090
C06853=1161.548,15.687,-47.666,-179.999,6.070,149.090
C06854=1161.553,15.437,-47.652,179.999,6.069,149.091
C06855=1161.559,15.188,-47.638,179.996,6.068,149.092
C06856=1161.564,14.939,-47.624,179.994,6.068,149.092
C06857=1161.569,14.689,-47.610,179.991,6.066,149.093
C06858=1161.574,14.439,-47.595,179.988,6.066,149.093
C06859=1161.579,14.190,-47.582,179.986,6.065,149.094
C06860=1161.585,13.940,-47.568,179.983,6.065,149.095
C06861=1161.590,13.690,-47.554,179.981,6.064,149.095
C06862=1161.594,13.441,-47.540,179.978,6.063,149.096
C06863=1161.599,13.192,-47.526,179.976,6.062,149.096
C06864=1161.604,12.942,-47.512,179.973,6.061,149.097
C06865=1161.609,12.692,-47.498,179.971,6.060,149.097
C06866=1161.615,12.443,-47.484,179.968,6.060,149.098
C06867=1161.620,12.193,-47.470,179.966,6.059,149.098
C06868=1161.625,11.943,-47.456,179.963,6.059,149.099
C06869=1161.630,11.695,-47.442,179.960,6.057,149.100
C06870=1161.635,11.445,-47.428,179.958,6.057,149.100
C06871=1161.640,11.195,-47.414,179.955,6.056,149.101
C06872=1161.646,10.946,-47.401,179.953,6.055,149.101
C06873=1161.651,10.696,-47.386,179.950,6.055,149.102
C06874=1161.656,10.446,-47.372,179.948,6.054,149.103
C06875=1161.660,10.197,-47.359,179.946,6.054,149.103
C06876=1161.666,9.947,-47.345,179.943,6.052,149.104
C06877=1161.671,9.697,-47.331,179.940,6.051,149.104
C06878=1161.676,9.448,-47.317,179.938,6.051,149.105
C06879=1161.681,9.199,-47.303,179.935,6.050,149.105
C06880=1161.686,8.949,-47.290,179.933,6.050,149.106
C06881=1161.691,8.700,-47.276,179.930,6.049,149.107
C06882=1161.696,8.450,-47.262,179.928,6.048,149.107
C06883=1161.702,8.200,-47.248,179.925,6.047,149.108
C06884=1161.706,7.951,-47.235,179.922,6.046,149.108
C06885=1161.711,7.701,-47.220,179.920,6.045,149.109
C06886=1161.717,7.452,-47.207,179.918,6.045,149.110
C06887=1161.722,7.202,-47.193,179.915,6.044,149.110
C06888=1161.727,6.953,-47.180,179.913,6.044,149.111
C06889=1161.732,6.703,-47.166,179.910,6.043,149.111
C06890=1161.737,6.453,-47.152,179.908,6.042,149.112
C06891=1161.742,6.204,-47.139,179.905,6.041,149.113
C06892=1161.747,5.954,-47.125,179.903,6.040,149.113
C06893=1161.753,5.705,-47.111,179.900,6.040,149.114
C06894=1161.758,5.455,-47.098,179.898,6.039,149.114
C06895=1161.762,5.205,-47.084,179.895,6.039,149.115
C06896=1161.768,4.956,-47.071,179.893,6.038,149.115
C06897=1161.773,4.706,-47.056,179.890,6.037,149.116
C06898=1161.778,4.457,-47.043,179.888,6.037,149.116
C06899=1161.783,4.207,-47.029,179.885,6.036,149.117
C06900=1161.789,3.958,-47.016,179.882,6.035,149.118
C06901=1161.793,3.708,-47.003,179.880,6.034,149.118
C06902=1161.798,3.458,-46.988,179.877,6.034,149.119
C06903=1161.803,3.209,-46.976,179.875,6.033,149.119
C06904=1161.808,2.959,-46.961,179.872,6.032,149.120
C06905=1161.814,2.710,-46.948,179.870,6.031,149.121
C06906=1161.818,2.460,-46.935,179.868,6.031,149.121
C06907=1161.825,2.191,-46.921,179.865,6.031,149.122
C06908=1161.830,1.921,-46.906,179.862,6.029,149.122
C06909=1161.835,1.652,-46.891,179.860,6.028,149.123
C06910=1161.840,1.382,-46.877,179.857,6.028,149.124
C06911=1161.846,1.133,-46.863,179.855,6.027,149.124
C06912=1161.851,0.883,-46.850,179.852,6.027,149.125
C06913=1161.856,0.634,-46.836,179.849,6.026,149.126
C06914=1161.861,0.384,-46.823,179.847,6.025,149.126
C06915=1161.866,0.135,-46.809,179.844,6.024,149.127
C06916=1161.871,-0.115,-46.796,179.842,6.023,149.127
C06917=1161.876,-0.364,-46.783,179.839,6.023,149.128
C06918=1161.881,-0.614,-46.769,179.837,6.022,149.128
C06919=1161.887,-0.864,-46.756,179.834,6.022,149.129
C06920=1161.892,-1.114,-46.743,179.832,6.021,149.130
C06921=1161.897,-1.363,-46.729,179.830,6.020,149.130
C06922=1161.903,-1.612,-46.716,179.827,6.020,149.131
C06923=1161.908,-1.862,-46.703,179.825,6.019,149.131
C06924=1161.913,-2.111,-46.689,179.822,6.019,149.132
C06925=1161.918,-2.361,-46.676,179.820,6.018,149.133
C06926=1161.923,-2.611,-46.663,179.817,6.017,149.133
C06927=1161.928,-2.860,-46.649,179.814,6.016,149.134
C06928=1161.933,-3.110,-46.636,179.812,6.015,149.134
C06929=1161.938,-3.360,-46.623,179.810,6.014,149.135
C06930=1161.943,-3.609,-46.609,179.807,6.014,149.136
C06931=1161.949,-3.858,-46.596,179.804,6.014,149.136
C06932=1161.954,-4.108,-46.583,179.802,6.013,149.137
C06933=1161.959,-4.358,-46.570,179.799,6.012,149.137
C06934=1161.964,-4.608,-46.556,179.797,6.011,149.138
C06935=1161.969,-4.857,-46.544,179.795,6.011,149.139
C06936=1161.974,-5.107,-46.530,179.792,6.010,149.139
C06937=1161.979,-5.356,-46.518,179.790,6.010,149.140
C06938=1161.985,-5.605,-46.504,179.788,6.009,149.140
C06939=1161.989,-5.856,-46.491,179.785,6.009,149.141
C06940=1161.995,-6.105,-46.478,179.782,6.008,149.142
C06941=1162.000,-6.355,-46.465,179.780,6.007,149.142
C06942=1162.005,-6.604,-46.452,179.778,6.007,149.143
C06943=1162.010,-6.853,-46.438,179.775,6.006,149.143
C06944=1162.015,-7.104,-46.425,179.772,6.005,149.144
C06945=1162.021,-7.353,-46.412,179.770,6.004,149.144
C06946=1162.026,-7.602,-46.399,179.767,6.003,149.145
C06947=1162.030,-7.852,-46.386,179.765,6.003,149.146
C06948=1162.036,-8.102,-46.373,179.762,6.002,149.146
C06949=1162.041,-8.352,-46.360,179.760,6.002,149.147
C06950=1162.046,-8.601,-46.348,179.758,6.001,149.147
C06951=1162.051,-8.850,-46.334,179.755,6.000,149.148
C06952=1162.056,-9.100,-46.321,179.753,6.000,149.149
C06953=1162.061,-9.350,-46.308,179.750,5.999,149.149
C06954=1162.067,-9.599,-46.295,179.748,5.998,149.150
C06955=1162.071,-9.849,-46.282,179.745,5.998,149.150
C06956=1162.076,-10.099,-46.269,179.743,5.998,149.151
C06957=1162.082,-10.348,-46.256,179.740,5.997,149.152
C06958=1162.087,-10.598,-46.243,179.738,5.996,149.152
C06959=1162.092,-10.848,-46.231,179.736,5.995,149.153
C06960=1162.098,-11.097,-46.217,179.733,5.995,149.153
C06961=1162.102,-11.347,-46.204,179.731,5.994,149.154
C06962=1162.108,-11.597,-46.192,179.728,5.994,149.155
C06963=1162.113,-11.846,-46.179,179.726,5.993,149.155
C06964=1162.118,-12.096,-46.166,179.723,5.992,149.156
C06965=1162.123,-12.346,-46.153,179.721,5.992,149.156
C06966=1162.128,-12.595,-46.140,179.718,5.991,149.157
C06967=1162.133,-12.844,-46.128,179.716,5.991,149.158
C06968=1162.139,-13.095,-46.114,179.714,5.990,149.158
C06969=1162.144,-13.344,-46.102,179.711,5.990,149.159
C06970=1162.149,-13.593,-46.089,179.709,5.989,149.159
C06971=1162.153,-13.843,-46.076,179.706,5.988,149.160
C06972=1162.159,-14.093,-46.063,179.704,5.987,149.160
C06973=1162.164,-14.342,-46.050,179.701,5.987,149.161
C06974=1162.169,-14.592,-46.038,179.699,5.987,149.162
C06975=1162.174,-14.842,-46.025,179.696,5.986,149.162
C06976=1162.180,-15.091,-46.012,179.694,5.985,149.163
C06977=1162.185,-15.340,-45.999,179.692,5.985,149.163
C06978=1162.190,-15.590,-45.987,179.689,5.984,149.164
C06979=1162.195,-15.840,-45.974,179.687,5.983,149.165
C06980=1162.200,-16.090,-45.961,179.684,5.983,149.165
C06981=1162.205,-16.339,-45.949,179.681,5.982,149.166
C06982=1162.211,-16.589,-45.936,179.679,5.982,149.166
C06983=1162.215,-16.839,-45.923,179.677,5.981,149.167
C06984=1162.221,-17.088,-45.910,179.674,5.980,149.168
C06985=1162.226,-17.338,-45.898,179.672,5.980,149.168
C06986=1162.231,-17.587,-45.886,179.670,5.979,149.169
C06987=1162.236,-17.837,-45.873,179.667,5.979,149.169
C06988=1162.242,-18.087,-45.859,179.665,5.978,149.170
C06989=1162.247,-18.336,-45.847,179.662,5.977,149.171
C06990=1162.252,-18.586,-45.835,179.659,5.977,149.171
C06991=1162.257,-18.836,-45.822,179.657,5.976,149.172
C06992=1162.262,-19.085,-45.810,179.655,5.976,149.172
C06993=1162.267,-19.335,-45.797,179.652,5.975,149.173
C06994=1162.272,-19.585,-45.785,179.650,5.974,149.174
C06995=1162.277,-19.834,-45.772,179.648,5.974,149.174
C06996=1162.283,-20.083,-45.760,179.645,5.973,149.175
C06997=1162.288,-20.333,-45.747,179.643,5.972,149.175
C06998=1162.294,-20.583,-45.735,179.640,5.972,149.176
C06999=1162.298,-20.833,-45.722,179.637,5.972,149.177
C07000=1162.303,-21.082,-45.709,179.635,5.971,149.177
C07001=1162.309,-21.332,-45.696,179.633,5.970,149.178
C07002=1162.314,-21.582,-45.685,179.630,5.969,149.178
C07003=1162.319,-21.831,-45.672,179.628,5.969,149.179
C07004=1162.324,-22.080,-45.659,179.626,5.968,149.179
C07005=1162.329,-22.331,-45.647,179.623,5.968,149.180
C07006=1162.334,-22.580,-45.635,179.621,5.968,149.181
C07007=1162.339,-22.829,-45.622,179.619,5.967,149.181
C07008=1162.345,-23.079,-45.610,179.616,5.967,149.182
C07009=1162.350,-23.329,-45.597,179.614,5.966,149.182
C07010=1162.355,-23.579,-45.586,179.611,5.966,149.183
C07011=1162.361,-23.849,-45.571,179.609,5.965,149.184
C07012=1162.367,-24.118,-45.559,179.606,5.964,149.184
C07013=1162.372,-24.388,-45.545,179.603,5.963,149.185
C07014=1162.377,-24.658,-45.532,179.600,5.963,149.186
C07015=1162.382,-24.908,-45.519,179.598,5.962,149.186
C07016=1162.388,-25.157,-45.507,179.596,5.962,149.187
C07017=1162.393,-25.407,-45.495,179.593,5.961,149.187
C07018=1162.398,-25.656,-45.482,179.591,5.960,149.188
C07019=1162.404,-25.906,-45.470,179.589,5.960,149.188
C07020=1162.409,-26.156,-45.458,179.586,5.960,149.189
C07021=1162.414,-26.406,-45.446,179.584,5.959,149.190
C07022=1162.419,-26.655,-45.433,179.582,5.959,149.190
C07023=1162.424,-26.905,-45.421,179.579,5.958,149.191
C07024=1162.429,-27.155,-45.409,179.577,5.957,149.192
C07025=1162.435,-27.405,-45.397,179.574,5.957,149.192
C07026=1162.440,-27.654,-45.384,179.572,5.956,149.193
C07027=1162.445,-27.904,-45.372,179.569,5.956,149.193
C07028=1162.450,-28.153,-45.360,179.567,5.955,149.194
C07029=1162.456,-28.403,-45.348,179.564,5.954,149.195
C07030=1162.460,-28.652,-45.336,179.562,5.954,149.195
C07031=1162.466,-28.902,-45.324,179.560,5.953,149.196
C07032=1162.471,-29.152,-45.311,179.557,5.953,149.196
C07033=1162.476,-29.401,-45.299,179.555,5.953,149.197
C07034=1162.481,-29.651,-45.287,179.553,5.952,149.198
C07035=1162.487,-29.901,-45.275,179.551,5.952,149.198
C07036=1162.492,-30.150,-45.262,179.548,5.951,149.199
C07037=1162.497,-30.400,-45.250,179.546,5.950,149.199
C07038=1162.502,-30.650,-45.239,179.543,5.950,149.200
C07039=1162.507,-30.899,-45.226,179.540,5.949,149.201
C07040=1162.512,-31.149,-45.215,179.538,5.949,149.201
C07041=1162.518,-31.399,-45.203,179.535,5.948,149.202
C07042=1162.523,-31.648,-45.190,179.533,5.947,149.202
C07043=1162.528,-31.898,-45.178,179.531,5.947,149.203
C07044=1162.533,-32.147,-45.166,179.528,5.946,149.203
C07045=1162.538,-32.397,-45.154,179.526,5.947,149.204
C07046=1162.544,-32.647,-45.142,179.524,5.946,149.205
C07047=1162.549,-32.896,-45.130,179.522,5.945,149.205
C07048=1162.554,-33.146,-45.118,179.519,5.945,149.206
C07049=1162.559,-33.396,-45.107,179.517,5.944,149.206
C07050=1162.564,-33.645,-45.094,179.514,5.944,149.207
C07051=1162.569,-33.895,-45.082,179.512,5.943,149.208
C07052=1162.575,-34.145,-45.070,179.509,5.942,149.208
C07053=1162.580,-34.395,-45.058,179.507,5.942,149.209
C07054=1162.585,-34.644,-45.046,179.504,5.941,149.210
C07055=1162.590,-34.894,-45.034,179.503,5.941,149.210
C07056=1162.596,-35.144,-45.023,179.500,5.941,149.211
C07057=1162.601,-35.393,-45.010,179.498,5.940,149.211
C07058=1162.605,-35.643,-44.999,179.495,5.940,149.212
C07059=1162.611,-35.893,-44.987,179.493,5.939,149.212
C07060=1162.616,-36.143,-44.975,179.490,5.938,149.213
C07061=1162.622,-36.393,-44.963,179.488,5.938,149.214
C07062=1162.626,-36.642,-44.951,179.486,5.937,149.214
C07063=1162.632,-36.891,-44.940,179.484,5.938,149.215
C07064=1162.638,-37.141,-44.928,179.481,5.937,149.215
C07065=1162.642,-37.390,-44.916,179.479,5.936,149.216
C07066=1162.648,-37.640,-44.904,179.476,5.935,149.217
C07067=1162.653,-37.890,-44.892,179.474,5.935,149.217
C07068=1162.657,-38.139,-44.881,179.472,5.934,149.218
C07069=1162.663,-38.389,-44.869,179.469,5.934,149.218
C07070=1162.668,-38.639,-44.857,179.467,5.933,149.219
C07071=1162.674,-38.889,-44.845,179.465,5.933,149.220
C07072=1162.678,-39.139,-44.834,179.462,5.933,149.220
C07073=1162.684,-39.387,-44.821,179.460,5.932,149.221
C07074=1162.690,-39.637,-44.810,179.457,5.932,149.221
C07075=1162.694,-39.887,-44.798,179.455,5.931,149.222
C07076=1162.700,-40.137,-44.786,179.452,5.931,149.223
C07077=1162.704,-40.386,-44.775,179.450,5.930,149.223
C07078=1162.710,-40.636,-44.763,179.447,5.929,149.224
C07079=1162.715,-40.886,-44.751,179.446,5.929,149.224
C07080=1162.720,-41.136,-44.740,179.443,5.929,149.225
C07081=1162.726,-41.385,-44.728,179.441,5.928,149.225
C07082=1162.731,-41.635,-44.717,179.438,5.928,149.226
C07083=1162.736,-41.885,-44.705,179.436,5.927,149.227
C07084=1162.742,-42.135,-44.693,179.434,5.926,149.227
C07085=1162.746,-42.384,-44.681,179.431,5.926,149.228
C07086=1162.751,-42.634,-44.670,179.429,5.926,149.229
C07087=1162.757,-42.883,-44.658,179.427,5.926,149.229
C07088=1162.762,-43.132,-44.647,179.424,5.925,149.230
C07089=1162.767,-43.382,-44.635,179.422,5.924,149.230
C07090=1162.772,-43.632,-44.624,179.420,5.924,149.231
C07091=1162.778,-43.882,-44.612,179.417,5.923,149.232
C07092=1162.782,-44.132,-44.600,179.415,5.923,149.232
C07093=1162.788,-44.381,-44.589,179.413,5.923,149.233
C07094=1162.793,-44.630,-44.578,179.410,5.922,149.233
C07095=1162.798,-44.880,-44.566,179.408,5.922,149.234
C07096=1162.804,-45.131,-44.555,179.406,5.921,149.234
C07097=1162.809,-45.381,-44.543,179.403,5.920,149.235
C07098=1162.815,-45.630,-44.532,179.401,5.920,149.236
C07099=1162.820,-45.879,-44.520,179.399,5.920,149.236
C07100=1162.825,-46.129,-44.509,179.396,5.920,149.237
C07101=1162.830,-46.379,-44.497,179.394,5.919,149.237
C07102=1162.835,-46.629,-44.485,179.391,5.918,149.238
C07103=1162.840,-46.878,-44.474,179.389,5.918,149.239
C07104=1162.846,-47.128,-44.463,179.386,5.917,149.239
C07105=1162.851,-47.377,-44.451,179.385,5.917,149.240
C07106=1162.856,-47.627,-44.439,179.382,5.917,149.241
C07107=1162.861,-47.876,-44.428,179.380,5.916,149.241
C07108=1162.867,-48.127,-44.417,179.377,5.915,149.242
C07109=1162.872,-48.376,-44.406,179.375,5.915,149.242
C07110=1162.876,-48.626,-44.395,179.373,5.915,149.243
C07111=1162.882,-48.875,-44.383,179.371,5.914,149.243
C07112=1162.887,-49.125,-44.372,179.368,5.914,149.244
C07113=1162.893,-49.375,-44.360,179.366,5.913,149.245
C07114=1162.898,-49.625,-44.349,179.363,5.913,149.245
C07115=1162.903,-49.895,-44.337,179.361,5.912,149.246
C07116=1162.909,-50.166,-44.325,179.358,5.911,149.246
C07117=1162.915,-50.437,-44.312,179.356,5.911,149.247
C07118=1162.921,-50.706,-44.300,179.353,5.911,149.248
C07119=1162.926,-50.957,-44.289,179.351,5.911,149.248
C07120=1162.931,-51.207,-44.277,179.349,5.910,149.249
C07121=1162.936,-51.455,-44.266,179.347,5.909,149.250
C07122=1162.941,-51.705,-44.255,179.344,5.909,149.250
C07123=1162.947,-51.956,-44.244,179.342,5.908,149.251
C07124=1162.952,-52.205,-44.233,179.340,5.909,149.251
C07125=1162.957,-52.455,-44.221,179.338,5.908,149.252
C07126=1162.962,-52.704,-44.210,179.335,5.907,149.253
C07127=1162.967,-52.954,-44.199,179.332,5.907,149.253
C07128=1162.973,-53.204,-44.188,179.330,5.906,149.254
C07129=1162.978,-53.453,-44.176,179.328,5.907,149.254
C07130=1162.983,-53.703,-44.166,179.326,5.906,149.255
C07131=1162.989,-53.953,-44.154,179.323,5.905,149.256
C07132=1162.994,-54.202,-44.143,179.321,5.905,149.256
C07133=1162.999,-54.453,-44.132,179.318,5.904,149.257
C07134=1163.005,-54.702,-44.121,179.317,5.904,149.257
C07135=1163.009,-54.951,-44.110,179.314,5.904,149.258
C07136=1163.014,-55.202,-44.099,179.312,5.903,149.258
C07137=1163.020,-55.451,-44.088,179.309,5.903,149.259
C07138=1163.025,-55.701,-44.076,179.307,5.902,149.260
C07139=1163.030,-55.951,-44.066,179.305,5.902,149.260
C07140=1163.035,-56.200,-44.055,179.303,5.901,149.261
C07141=1163.041,-56.450,-44.043,179.300,5.901,149.262
C07142=1163.046,-56.700,-44.032,179.298,5.900,149.262
C07143=1163.051,-56.949,-44.021,179.296,5.901,149.263
C07144=1163.057,-57.199,-44.010,179.294,5.900,149.263
C07145=1163.062,-57.448,-43.999,179.291,5.899,149.264
C07146=1163.067,-57.698,-43.988,179.289,5.899,149.264
C07147=1163.072,-57.948,-43.977,179.286,5.898,149.265
C07148=1163.078,-58.197,-43.966,179.284,5.898,149.266
C07149=1163.083,-58.448,-43.955,179.282,5.898,149.266
C07150=1163.088,-58.697,-43.944,179.280,5.897,149.267
C07151=1163.093,-58.947,-43.934,179.277,5.897,149.267
C07152=1163.098,-59.196,-43.923,179.275,5.897,149.268
C07153=1163.104,-59.446,-43.911,179.273,5.896,149.269
C07154=1163.109,-59.696,-43.900,179.270,5.895,149.269
C07155=1163.114,-59.946,-43.889,179.268,5.895,149.270
C07156=1163.119,-60.195,-43.879,179.266,5.894,149.270
C07157=1163.125,-60.445,-43.867,179.264,5.895,149.271
C07158=1163.130,-60.695,-43.857,179.261,5.894,149.271
C07159=1163.135,-60.944,-43.846,179.259,5.893,149.272
C07160=1163.140,-61.194,-43.835,179.256,5.893,149.273
C07161=1163.145,-61.443,-43.824,179.254,5.893,149.273
C07162=1163.150,-61.694,-43.813,179.252,5.892,149.274
C07163=1163.156,-61.943,-43.803,179.250,5.892,149.275
C07164=1163.161,-62.193,-43.791,179.247,5.891,149.275
C07165=1163.167,-62.443,-43.781,179.245,5.891,149.276
C07166=1163.171,-62.692,-43.770,179.243,5.891,149.276
C07167=1163.177,-62.942,-43.760,179.240,5.890,149.277
C07168=1163.182,-63.191,-43.748,179.238,5.889,149.277
C07169=1163.187,-63.442,-43.737,179.236,5.890,149.278
C07170=1163.193,-63.692,-43.727,179.234,5.889,149.279
C07171=1163.198,-63.941,-43.716,179.231,5.889,149.279
C07172=1163.203,-64.191,-43.705,179.229,5.888,149.280
C07173=1163.208,-64.440,-43.694,179.227,5.888,149.280
C07174=1163.214,-64.690,-43.684,179.225,5.887,149.281
C07175=1163.219,-64.940,-43.673,179.222,5.887,149.282
C07176=1163.224,-65.189,-43.662,179.220,5.886,149.282
C07177=1163.229,-65.439,-43.652,179.218,5.887,149.283
C07178=1163.235,-65.689,-43.641,179.216,5.886,149.283
C07179=1163.240,-65.939,-43.630,179.213,5.885,149.284
C07180=1163.246,-66.188,-43.620,179.211,5.885,149.285
C07181=1163.251,-66.439,-43.609,179.209,5.885,149.285
C07182=1163.256,-66.687,-43.598,179.207,5.884,149.286
C07183=1163.261,-66.938,-43.588,179.204,5.884,149.286
C07184=1163.266,-67.187,-43.577,179.202,5.884,149.287
C07185=1163.271,-67.437,-43.566,179.200,5.883,149.288
C07186=1163.277,-67.686,-43.556,179.198,5.883,149.288
C07187=1163.282,-67.937,-43.545,179.195,5.882,149.289
C07188=1163.287,-68.186,-43.534,179.193,5.882,149.289
C07189=1163.292,-68.436,-43.524,179.191,5.882,149.290
C07190=1163.298,-68.685,-43.514,179.188,5.881,149.290
C07191=1163.303,-68.936,-43.503,179.186,5.880,149.291
C07192=1163.308,-69.185,-43.492,179.184,5.881,149.292
C07193=1163.314,-69.434,-43.482,179.182,5.880,149.292
C07194=1163.319,-69.684,-43.471,179.179,5.880,149.293
C07195=1163.325,-69.934,-43.460,179.178,5.880,149.293
C07196=1163.330,-70.184,-43.450,179.175,5.879,149.294
C07197=1163.335,-70.433,-43.439,179.173,5.878,149.294
C07198=1163.340,-70.684,-43.428,179.170,5.878,149.295
C07199=1163.346,-70.933,-43.418,179.169,5.878,149.296
C07200=1163.351,-71.183,-43.408,179.166,5.878,149.296
C07201=1163.356,-71.433,-43.398,179.164,5.877,149.297
C07202=1163.361,-71.682,-43.387,179.162,5.877,149.298
C07203=1163.366,-71.932,-43.377,179.159,5.876,149.298
C07204=1163.371,-72.181,-43.366,179.157,5.876,149.299
C07205=1163.376,-72.432,-43.356,179.155,5.875,149.299
C07206=1163.382,-72.681,-43.346,179.152,5.876,149.300
C07207=1163.388,-72.931,-43.335,179.150,5.875,149.300
C07208=1163.392,-73.180,-43.324,179.148,5.874,149.301
C07209=1163.398,-73.430,-43.314,179.146,5.874,149.302
C07210=1163.403,-73.680,-43.303,179.144,5.874,149.302
C07211=1163.409,-73.930,-43.293,179.141,5.873,149.303
C07212=1163.414,-74.179,-43.283,179.139,5.873,149.303
C07213=1163.419,-74.429,-43.272,179.137,5.873,149.304
C07214=1163.425,-74.679,-43.262,179.135,5.872,149.304
C07215=1163.430,-74.929,-43.252,179.132,5.872,149.305
C07216=1163.435,-75.179,-43.241,179.130,5.872,149.306
C07217=1163.441,-75.428,-43.231,179.128,5.871,149.306
C07218=1163.446,-75.679,-43.220,179.126,5.871,149.307
C07219=1163.451,-75.949,-43.209,179.123,5.870,149.308
C07220=1163.457,-76.220,-43.198,179.121,5.871,149.308
C07221=1163.463,-76.491,-43.187,179.119,5.870,149.309
C07222=1163.469,-76.762,-43.176,179.116,5.869,149.309
C07223=1163.473,-77.012,-43.166,179.114,5.869,149.310
C07224=1163.479,-77.262,-43.155,179.112,5.869,149.311
C07225=1163.485,-77.511,-43.145,179.110,5.868,149.311
C07226=1163.490,-77.762,-43.135,179.107,5.868,149.312
C07227=1163.495,-78.011,-43.124,179.105,5.868,149.312
C07228=1163.501,-78.261,-43.114,179.103,5.867,149.313
C07229=1163.506,-78.511,-43.104,179.100,5.867,149.314
C07230=1163.511,-78.760,-43.093,179.098,5.866,149.314
C07231=1163.516,-79.010,-43.084,179.096,5.866,149.315
C07232=1163.521,-79.260,-43.073,179.094,5.866,149.315
C07233=1163.527,-79.509,-43.063,179.091,5.865,149.316
C07234=1163.532,-79.759,-43.053,179.090,5.865,149.316
C07235=1163.537,-80.009,-43.042,179.087,5.865,149.317
C07236=1163.543,-80.259,-43.033,179.085,5.864,149.318
C07237=1163.548,-80.509,-43.023,179.083,5.864,149.318
C07238=1163.554,-80.758,-43.013,179.081,5.864,149.319
C07239=1163.559,-81.008,-43.002,179.078,5.863,149.319
C07240=1163.564,-81.258,-42.992,179.076,5.863,149.320
C07241=1163.569,-81.507,-42.982,179.074,5.862,149.320
C07242=1163.574,-81.757,-42.972,179.071,5.862,149.321
C07243=1163.580,-82.007,-42.962,179.070,5.862,149.322
C07244=1163.585,-82.257,-42.951,179.067,5.862,149.322
C07245=1163.590,-82.506,-42.942,179.065,5.861,149.323
C07246=1163.596,-82.757,-42.932,179.063,5.861,149.324
C07247=1163.601,-83.006,-42.922,179.061,5.861,149.324
C07248=1163.607,-83.256,-42.912,179.058,5.860,149.325
C07249=1163.611,-83.506,-42.902,179.056,5.860,149.325
C07250=1163.617,-83.755,-42.891,179.054,5.859,149.326
C07251=1163.622,-84.005,-42.881,179.052,5.859,149.326
C07252=1163.627,-84.255,-42.872,179.050,5.859,149.327
C07253=1163.632,-84.505,-42.862,179.047,5.859,149.328
C07254=1163.638,-84.754,-42.852,179.045,5.858,149.328
C07255=1163.644,-85.004,-42.841,179.044,5.858,149.329
C07256=1163.648,-85.253,-42.832,179.041,5.858,149.329
C07257=1163.653,-85.503,-42.821,179.039,5.858,149.330
C07258=1163.659,-85.754,-42.812,179.037,5.857,149.330
C07259=1163.664,-86.003,-42.802,179.034,5.856,149.331
C07260=1163.670,-86.252,-42.792,179.032,5.857,149.332
C07261=1163.675,-86.502,-42.782,179.030,5.856,149.332
C07262=1163.680,-86.752,-42.772,179.028,5.855,149.333
C07263=1163.686,-87.002,-42.762,179.026,5.856,149.333
C07264=1163.691,-87.252,-42.752,179.024,5.855,149.334
C07265=1163.696,-87.501,-42.742,179.021,5.854,149.335
C07266=1163.701,-87.752,-42.732,179.019,5.854,149.335
C07267=1163.707,-88.001,-42.722,179.017,5.854,149.336
C07268=1163.712,-88.250,-42.713,179.014,5.853,149.336
C07269=1163.718,-88.501,-42.703,179.013,5.853,149.337
C07270=1163.723,-88.750,-42.694,179.010,5.853,149.337
C07271=1163.728,-89.000,-42.683,179.009,5.853,149.338
C07272=1163.733,-89.250,-42.673,179.006,5.853,149.339
C07273=1163.738,-89.499,-42.664,179.004,5.852,149.339
C07274=1163.744,-89.749,-42.654,179.002,5.852,149.340
C07275=1163.749,-89.999,-42.643,179.000,5.851,149.340
C07276=1163.755,-90.248,-42.635,178.997,5.851,149.341
C07277=1163.760,-90.499,-42.624,178.995,5.851,149.341
C07278=1163.765,-90.748,-42.614,178.993,5.850,149.342
C07279=1163.770,-90.998,-42.605,178.990,5.850,149.343
C07280=1163.775,-91.247,-42.595,178.989,5.850,149.343
C07281=1163.781,-91.497,-42.586,178.987,5.849,149.344
C07282=1163.787,-91.747,-42.576,178.985,5.850,149.344
C07283=1163.791,-91.997,-42.566,178.982,5.849,149.345
C07284=1163.797,-92.247,-42.556,178.980,5.848,149.346
C07285=1163.802,-92.496,-42.546,178.978,5.848,149.346
C07286=1163.808,-92.746,-42.537,178.976,5.848,149.347
C07287=1163.813,-92.996,-42.527,178.974,5.848,149.347
C07288=1163.818,-93.245,-42.517,178.972,5.847,149.348
C07289=1163.824,-93.495,-42.508,178.969,5.847,149.348
C07290=1163.828,-93.745,-42.498,178.967,5.847,149.349
C07291=1163.834,-93.995,-42.488,178.965,5.846,149.349
C07292=1163.839,-94.245,-42.479,178.962,5.846,149.350
C07293=1163.845,-94.495,-42.469,178.961,5.846,149.351
C07294=1163.850,-94.744,-42.459,178.958,5.845,149.351
C07295=1163.856,-94.994,-42.450,178.957,5.845,149.352
C07296=1163.861,-95.244,-42.440,178.954,5.845,149.352
C07297=1163.866,-95.493,-42.430,178.952,5.844,149.353
C07298=1163.871,-95.743,-42.421,178.950,5.844,149.353
C07299=1163.876,-95.993,-42.411,178.948,5.844,149.354
C07300=1163.882,-96.243,-42.402,178.946,5.844,149.355
C07301=1163.887,-96.493,-42.392,178.944,5.843,149.355
C07302=1163.892,-96.742,-42.383,178.941,5.843,149.356
C07303=1163.898,-96.993,-42.373,178.939,5.843,149.356
C07304=1163.903,-97.242,-42.364,178.937,5.842,149.357
C07305=1163.909,-97.492,-42.354,178.935,5.842,149.358
C07306=1163.914,-97.741,-42.344,178.933,5.842,149.358
C07307=1163.919,-97.991,-42.336,178.930,5.841,149.359
C07308=1163.925,-98.241,-42.325,178.929,5.841,149.359
C07309=1163.930,-98.490,-42.316,178.926,5.841,149.360
C07310=1163.935,-98.740,-42.306,178.924,5.841,149.360
C07311=1163.941,-98.990,-42.297,178.922,5.840,149.361
C07312=1163.946,-99.240,-42.288,178.920,5.839,149.361
C07313=1163.951,-99.489,-42.278,178.918,5.840,149.362
C07314=1163.957,-99.740,-42.268,178.916,5.839,149.363
